// TIA Portal V20 export
// export: Created 2025-12-01T14:57:24.3574647Z, ExportSetting None, DisplayName Totally Integrated Automation Portal, DisplayVersion V20 Update 3, DisplayName TIA Portal Openness, DisplayVersion V20 Update 3, DisplayName TIA Portal Version Control Interface, DisplayVersion V20 Update 3, DisplayName STEP 7 Professional, DisplayVersion V20 Update 3, DisplayName STEP 7 Safety, DisplayVersion V20 Update 2, DisplayName WinCC Basic/Comfort/Advanced, DisplayVersion V20 Update 3, DisplayName WinCC Professional, DisplayVersion V20 Update 3, DisplayName WinCC Unified, DisplayVersion V20 Update 3
FUNCTION_BLOCK "FB20_M_PASO_E1E3_S1S3_2Puertas"   // FB20, LAD
TITLE = Control del Ramal de Salidas
{ S7_Optimized_Access := 'FALSE' }
AUTHOR : PASO
NAME : 20150327
VERSION : 3.3
// stored: AutoNumber false, SetENOAutomatically false
   VAR_INPUT
      Mesa : UInt;   // Mesa de la FB
      Error_Tx : Bool;
      EnTension : Bool;   // Existe Tension en la Mesa
      Termico_Tx : Bool;
      pHsMx_1 : Bool;   // Desactiva si Transferencia controlada
      pHsMx_2 : Bool;   // Desactiva si Transferencia controlada
      pHsMx_PR1 : Bool;   // pHs de Protrusion de la Mesa. Nota: No existe >> ON
      pHsMx_PR3 : Bool;   // pHs de Protrusion de la Mesa. Nota: No existe >> ON
      Avance_Tx : Bool;
      Retroceso_Tx : Bool;
      PUE1_Abierta : Bool;
      PUE1_Cerrada : Bool;
      PUE3_Abierta : Bool;
      PUE3_Cerrada : Bool;
      MAnt_DescargaAct_M1 : Bool;
      ATF_Ent_M1 : Bool;
      P_Mens_Ent_M1 : Bool;
      MAnt_DescargaAct_M3 : Bool;
      AVTF_Ent_M3 : Bool;
      P_Mens_Ent_M3 : Bool;
      PTF_Sal_M1 : Bool;
      FTF_Sal_M1 : Bool;
      PTF_Sal_M3 : Bool;
      FTF_Sal_M3 : Bool;
      Mx_VelocidadLenta_In : Bool;   // Forzar a Velociada Lenta
      F_EnvMens_Mx : Bool;
      OrdSal_S01 : Bool;
      OrdSal_S03 : Bool;
      V_CNT_pHsMx : Int := 300;
      V_CNT_pHsMx_FTF : Int := 50;   // Valor contador para FTF_Mant
      V_CNTSeg_pHsMx : Int := 2000;
      V_CNT_PasoLenta : Int := 2000;
      V_CNT_ApHsMx : Int := 500;
      V_CNTSeg_ApHsMx : Int := 2000;
      V_CNT_Simultaneo : Int := 1000;
      V_InicioSimultaneo : Int := 0;
      V_FinSimultaneo : Int := 0;
      V_TOut_Tx_Mx : Int := 30000;
      V_TOut_PUERTA : Int := 5000;
      V_TMP_Protrusion : Int := 200;   // TMP de Protrusion
      V_CNT_PerdidapHs : Int := 1000;
   END_VAR
   VAR_OUTPUT
      P_EnvMens_PMx : Bool;
      P_RecepOK_Mx : Bool;
      PTF_Ent_M1 : Bool;
      FTF_Ent_M1 : Bool;
      PTF_Ent_M3 : Bool;
      FTF_Ent_M3 : Bool;
      AVTF_Sal_M1 : Bool;
      P_Mens_Sal_M1 : Bool;
      AVTF_Sal_M3 : Bool;
      P_Mens_Sal_M3 : Bool;
   END_VAR
   VAR
      Anular_prE1 : Bool;   // ???
      Anular_prS3 : Bool;   // ???
      Mx_ET00 : Bool;
      Mx_ET01 : Bool;
      Mx_ET02 : Bool;
      Mx_ET08 : Bool;
      Mx_ET09 : Bool;
      Mx_ET10 : Bool;
      Mx_ET11 : Bool;
      Mx_ET12 : Bool;
      Mx_ET13 : Bool;
      Mx_ET50 : Bool;
      Mx_ET51 : Bool;
      Mx_ET110 : Bool;
      Mx_ET111 : Bool;
      Mx_ET150 : Bool;
      Mx_ET151 : Bool;
      Selec_M1_Entrada : Bool;
      Selec_M3_Entrada : Bool;
      Selec_M1_Salida : Bool;
      Selec_M3_Salida : Bool;
      MEnt_DescargaAct : Bool;
      AVTF_MEnt : Bool;
      P_Mens_MEnt : Bool;   // Interlock >> P_Mens de MAnt >> Mx
      PTF_MEnt : Bool;
      FTF_MEnt : Bool;
      AVTF_MSal : Bool;
      P_Mens_MSal : Bool;   // Interlock >> P_Mens de Mx >> MSig
      PTF_MSal : Bool;
      FTF_MSal : Bool;
      ProtocoloIniciado : Bool;
      CNT_pHsMx_FTF_OK : Bool;
      Simultaneo_Mx : Bool;
      STAT_EnvMens_PMx : Bool;
      MA_Abrir_PUE1 : Bool;
      MA_Cerrar_PUE1 : Bool;
      MA_Abrir_PUE3 : Bool;
      MA_Cerrar_PUE3 : Bool;
      CNT_pHsMx { S7_SetPoint := 'True'} : "FB910_CNT_UHS";
      CNTSeg_pHsMx { S7_SetPoint := 'True'} : "FB910_CNT_UHS";
      CNT_ApHsMx { S7_SetPoint := 'True'} : "FB910_CNT_UHS";
      CNTSeg_ApHsMx { S7_SetPoint := 'True'} : "FB910_CNT_UHS";
      CNT_Simultaneo { S7_SetPoint := 'True'} : "FB910_CNT_UHS";
      TMP_EnTension { S7_SetPoint := 'True'} : "FB910_CNT_UHS";
      TOut_Av_Mx { S7_SetPoint := 'True'} : "FB910_CNT_UHS";
      TOut_Ret_Mx { S7_SetPoint := 'True'} : "FB910_CNT_UHS";
      TOut_Abrir_PUE1 { S7_SetPoint := 'True'} : "FB910_CNT_UHS";
      TOut_Cerrar_PUE1 { S7_SetPoint := 'True'} : "FB910_CNT_UHS";
      TOut_Abrir_PUE3 { S7_SetPoint := 'True'} : "FB910_CNT_UHS";
      TOut_Cerrar_PUE3 { S7_SetPoint := 'True'} : "FB910_CNT_UHS";
      TMP_Protrusion { S7_SetPoint := 'True'} : "FB910_CNT_UHS";   // TMP de la Protrusion
      CNT_PerdidapHs { S7_SetPoint := 'True'} : "FB910_CNT_UHS";
   END_VAR
   VAR_TEMP
      EstadoZona : "EstadoZona";   // Estado de Zona de la Mesa
      EstadoVI : "EstadosMesa";   // Estado del Vehiculo Inteliguente de la Mesa
      ConfigFB : "UDT_ConfigFB";   // Configuracion de la FB de la Mesa
      V_Protrusion : Int;
      Aux_ET00 : Bool;
   END_VAR
   VAR_TEMP   // added for the SCL form of the ladder/FBD networks
      _w1 : Bool;
      _w2 : Bool;
   END_VAR
BEGIN

REGION Network 1: INICIALIZAR - Recoger las Variables de Estado de la Mesa
   // Se recoge - Estado_CBx
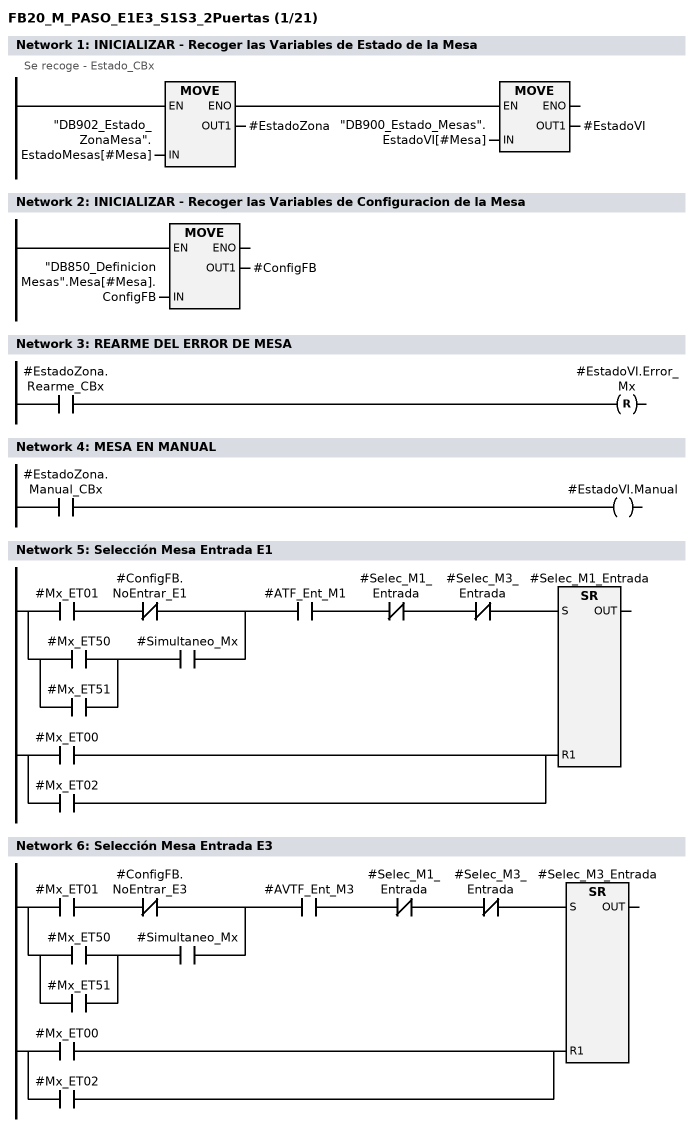
   RUNG wire#powerrail
      Move(in := "DB902_Estado_ZonaMesa".EstadoMesas[#Mesa], out1 => #EstadoZona)
      Move(in := "DB900_Estado_Mesas".EstadoVI[#Mesa], out1 => #EstadoVI)
   END_RUNG
   // the same network as SCL:
   #EstadoZona := "DB902_Estado_ZonaMesa".EstadoMesas[#Mesa];
   #EstadoVI := "DB900_Estado_Mesas".EstadoVI[#Mesa];
END_REGION

REGION Network 2: INICIALIZAR - Recoger las Variables de Configuracion de la Mesa
   RUNG wire#powerrail
      Move(in := "DB850_DefinicionMesas".Mesa[#Mesa].ConfigFB, out1 => #ConfigFB)
   END_RUNG
   // the same network as SCL:
   #ConfigFB := "DB850_DefinicionMesas".Mesa[#Mesa].ConfigFB;
END_REGION

REGION Network 3: REARME DEL ERROR DE MESA
   RUNG wire#powerrail
      Contact( #EstadoZona.Rearme_CBx )
      R_Coil( #EstadoVI.Error_Mx )
   END_RUNG
   // the same network as SCL:
   IF #EstadoZona.Rearme_CBx THEN #EstadoVI.Error_Mx := FALSE; END_IF;
END_REGION

REGION Network 4: MESA EN MANUAL
   RUNG wire#powerrail
      Contact( #EstadoZona.Manual_CBx )
      Coil( #EstadoVI.Manual )
   END_RUNG
   // the same network as SCL:
   #EstadoVI.Manual := #EstadoZona.Manual_CBx;
END_REGION

REGION Network 5: Selección Mesa Entrada E1
   RUNG wire#powerrail
      Contact( #Mx_ET01 )
      I_Contact( #ConfigFB.NoEntrar_E1 )
      wire#w1
      Contact( #ATF_Ent_M1 )
      I_Contact( #Selec_M1_Entrada )
      I_Contact( #Selec_M3_Entrada )
      S_SR(operand := #Selec_M1_Entrada, r1 := wire#w3)
   END_RUNG
   RUNG wire#powerrail
      Contact( #Mx_ET50 )
      wire#w2
      Contact( #Simultaneo_Mx )
   END_RUNG wire#w1
   RUNG wire#powerrail
      Contact( #Mx_ET51 )
   END_RUNG wire#w2
   RUNG wire#powerrail
      Contact( #Mx_ET00 )
   END_RUNG wire#w3
   RUNG wire#powerrail
      Contact( #Mx_ET02 )
   END_RUNG wire#w3
   // the same network as SCL:
   IF ((#Mx_ET01 AND NOT #ConfigFB.NoEntrar_E1) OR ((#Mx_ET50 OR #Mx_ET51) AND #Simultaneo_Mx)) AND #ATF_Ent_M1 AND NOT #Selec_M1_Entrada AND NOT #Selec_M3_Entrada THEN
       #Selec_M1_Entrada := TRUE;   // SR flip-flop
   END_IF;
   IF #Mx_ET00 OR #Mx_ET02 THEN #Selec_M1_Entrada := FALSE; END_IF;
END_REGION

REGION Network 6: Selección Mesa Entrada E3
   RUNG wire#powerrail
      Contact( #Mx_ET01 )
      I_Contact( #ConfigFB.NoEntrar_E3 )
      wire#w1
      Contact( #AVTF_Ent_M3 )
      I_Contact( #Selec_M1_Entrada )
      I_Contact( #Selec_M3_Entrada )
      S_SR(operand := #Selec_M3_Entrada, r1 := wire#w3)
   END_RUNG
   RUNG wire#powerrail
      Contact( #Mx_ET50 )
      wire#w2
      Contact( #Simultaneo_Mx )
   END_RUNG wire#w1
   RUNG wire#powerrail
      Contact( #Mx_ET51 )
   END_RUNG wire#w2
   RUNG wire#powerrail
      Contact( #Mx_ET00 )
   END_RUNG wire#w3
   RUNG wire#powerrail
      Contact( #Mx_ET02 )
   END_RUNG wire#w3
   // the same network as SCL:
   IF ((#Mx_ET01 AND NOT #ConfigFB.NoEntrar_E3) OR ((#Mx_ET50 OR #Mx_ET51) AND #Simultaneo_Mx)) AND #AVTF_Ent_M3 AND NOT #Selec_M1_Entrada AND NOT #Selec_M3_Entrada THEN
       #Selec_M3_Entrada := TRUE;   // SR flip-flop
   END_IF;
   IF #Mx_ET00 OR #Mx_ET02 THEN #Selec_M3_Entrada := FALSE; END_IF;
END_REGION

REGION Network 7: Selección Mesa Salida S1
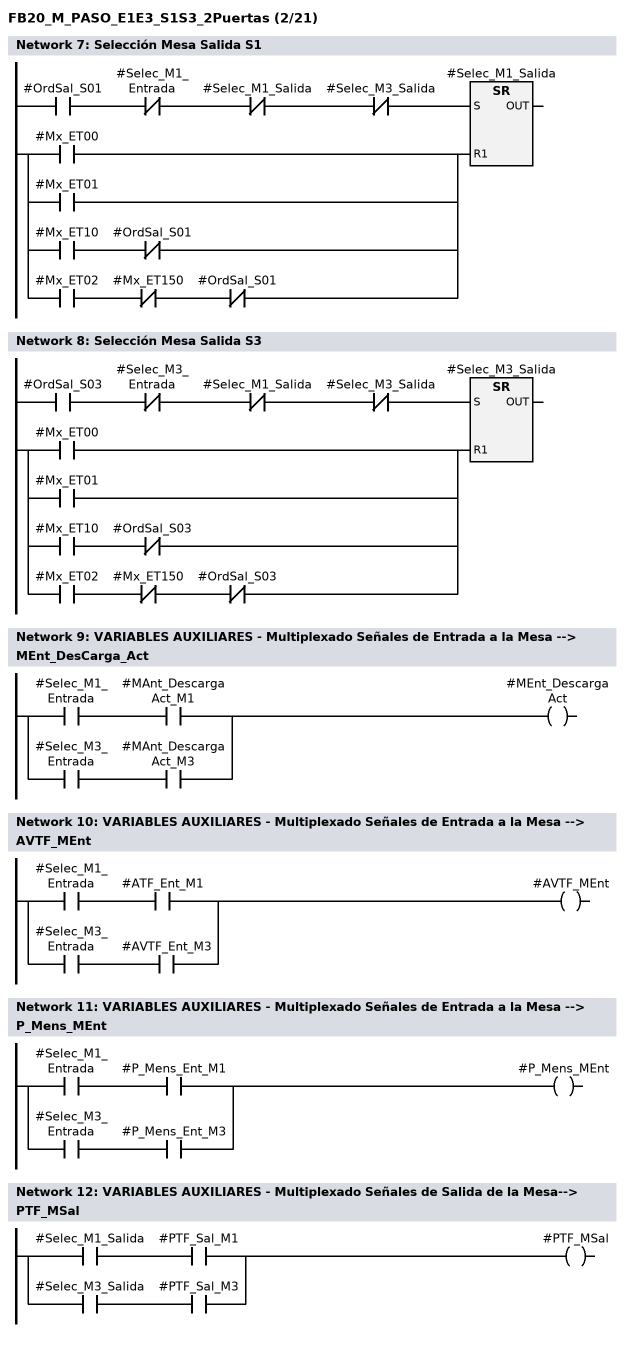
   RUNG wire#powerrail
      Contact( #OrdSal_S01 )
      I_Contact( #Selec_M1_Entrada )
      I_Contact( #Selec_M1_Salida )
      I_Contact( #Selec_M3_Salida )
      S_SR(operand := #Selec_M1_Salida, r1 := wire#w1)
   END_RUNG
   RUNG wire#powerrail
      Contact( #Mx_ET00 )
   END_RUNG wire#w1
   RUNG wire#powerrail
      Contact( #Mx_ET01 )
   END_RUNG wire#w1
   RUNG wire#powerrail
      Contact( #Mx_ET10 )
      I_Contact( #OrdSal_S01 )
   END_RUNG wire#w1
   RUNG wire#powerrail
      Contact( #Mx_ET02 )
      I_Contact( #Mx_ET150 )
      I_Contact( #OrdSal_S01 )
   END_RUNG wire#w1
   // the same network as SCL:
   IF #OrdSal_S01 AND NOT #Selec_M1_Entrada AND NOT #Selec_M1_Salida AND NOT #Selec_M3_Salida THEN
       #Selec_M1_Salida := TRUE;   // SR flip-flop
   END_IF;
   IF #Mx_ET00 OR #Mx_ET01 OR (#Mx_ET10 AND NOT #OrdSal_S01) OR (#Mx_ET02 AND NOT #Mx_ET150 AND NOT #OrdSal_S01) THEN
       #Selec_M1_Salida := FALSE;
   END_IF;
END_REGION

REGION Network 8: Selección Mesa Salida S3
   RUNG wire#powerrail
      Contact( #OrdSal_S03 )
      I_Contact( #Selec_M3_Entrada )
      I_Contact( #Selec_M1_Salida )
      I_Contact( #Selec_M3_Salida )
      S_SR(operand := #Selec_M3_Salida, r1 := wire#w1)
   END_RUNG
   RUNG wire#powerrail
      Contact( #Mx_ET00 )
   END_RUNG wire#w1
   RUNG wire#powerrail
      Contact( #Mx_ET01 )
   END_RUNG wire#w1
   RUNG wire#powerrail
      Contact( #Mx_ET10 )
      I_Contact( #OrdSal_S03 )
   END_RUNG wire#w1
   RUNG wire#powerrail
      Contact( #Mx_ET02 )
      I_Contact( #Mx_ET150 )
      I_Contact( #OrdSal_S03 )
   END_RUNG wire#w1
   // the same network as SCL:
   IF #OrdSal_S03 AND NOT #Selec_M3_Entrada AND NOT #Selec_M1_Salida AND NOT #Selec_M3_Salida THEN
       #Selec_M3_Salida := TRUE;   // SR flip-flop
   END_IF;
   IF #Mx_ET00 OR #Mx_ET01 OR (#Mx_ET10 AND NOT #OrdSal_S03) OR (#Mx_ET02 AND NOT #Mx_ET150 AND NOT #OrdSal_S03) THEN
       #Selec_M3_Salida := FALSE;
   END_IF;
END_REGION

REGION Network 9: VARIABLES AUXILIARES - Multiplexado Señales de Entrada a la Mesa --> MEnt_DesCarga_Act
   RUNG wire#powerrail
      Contact( #Selec_M1_Entrada )
      Contact( #MAnt_DescargaAct_M1 )
      wire#w1
      Coil( #MEnt_DescargaAct )
   END_RUNG
   RUNG wire#powerrail
      Contact( #Selec_M3_Entrada )
      Contact( #MAnt_DescargaAct_M3 )
   END_RUNG wire#w1
   // the same network as SCL:
   #MEnt_DescargaAct := (#Selec_M1_Entrada AND #MAnt_DescargaAct_M1) OR (#Selec_M3_Entrada AND #MAnt_DescargaAct_M3);
END_REGION

REGION Network 10: VARIABLES AUXILIARES - Multiplexado Señales de Entrada a la Mesa --> AVTF_MEnt
   RUNG wire#powerrail
      Contact( #Selec_M1_Entrada )
      Contact( #ATF_Ent_M1 )
      wire#w1
      Coil( #AVTF_MEnt )
   END_RUNG
   RUNG wire#powerrail
      Contact( #Selec_M3_Entrada )
      Contact( #AVTF_Ent_M3 )
   END_RUNG wire#w1
   // the same network as SCL:
   #AVTF_MEnt := (#Selec_M1_Entrada AND #ATF_Ent_M1) OR (#Selec_M3_Entrada AND #AVTF_Ent_M3);
END_REGION

REGION Network 11: VARIABLES AUXILIARES - Multiplexado Señales de Entrada a la Mesa --> P_Mens_MEnt
   RUNG wire#powerrail
      Contact( #Selec_M1_Entrada )
      Contact( #P_Mens_Ent_M1 )
      wire#w1
      Coil( #P_Mens_MEnt )
   END_RUNG
   RUNG wire#powerrail
      Contact( #Selec_M3_Entrada )
      Contact( #P_Mens_Ent_M3 )
   END_RUNG wire#w1
   // the same network as SCL:
   #P_Mens_MEnt := (#Selec_M1_Entrada AND #P_Mens_Ent_M1) OR (#Selec_M3_Entrada AND #P_Mens_Ent_M3);
END_REGION

REGION Network 12: VARIABLES AUXILIARES - Multiplexado Señales de Salida de la Mesa--> PTF_MSal
   RUNG wire#powerrail
      Contact( #Selec_M1_Salida )
      Contact( #PTF_Sal_M1 )
      wire#w1
      Coil( #PTF_MSal )
   END_RUNG
   RUNG wire#powerrail
      Contact( #Selec_M3_Salida )
      Contact( #PTF_Sal_M3 )
   END_RUNG wire#w1
   // the same network as SCL:
   #PTF_MSal := (#Selec_M1_Salida AND #PTF_Sal_M1) OR (#Selec_M3_Salida AND #PTF_Sal_M3);
END_REGION

REGION Network 13: VARIABLES AUXILIARES - Multiplexado Señales de Salida de la Mesa--> FTF_MSal
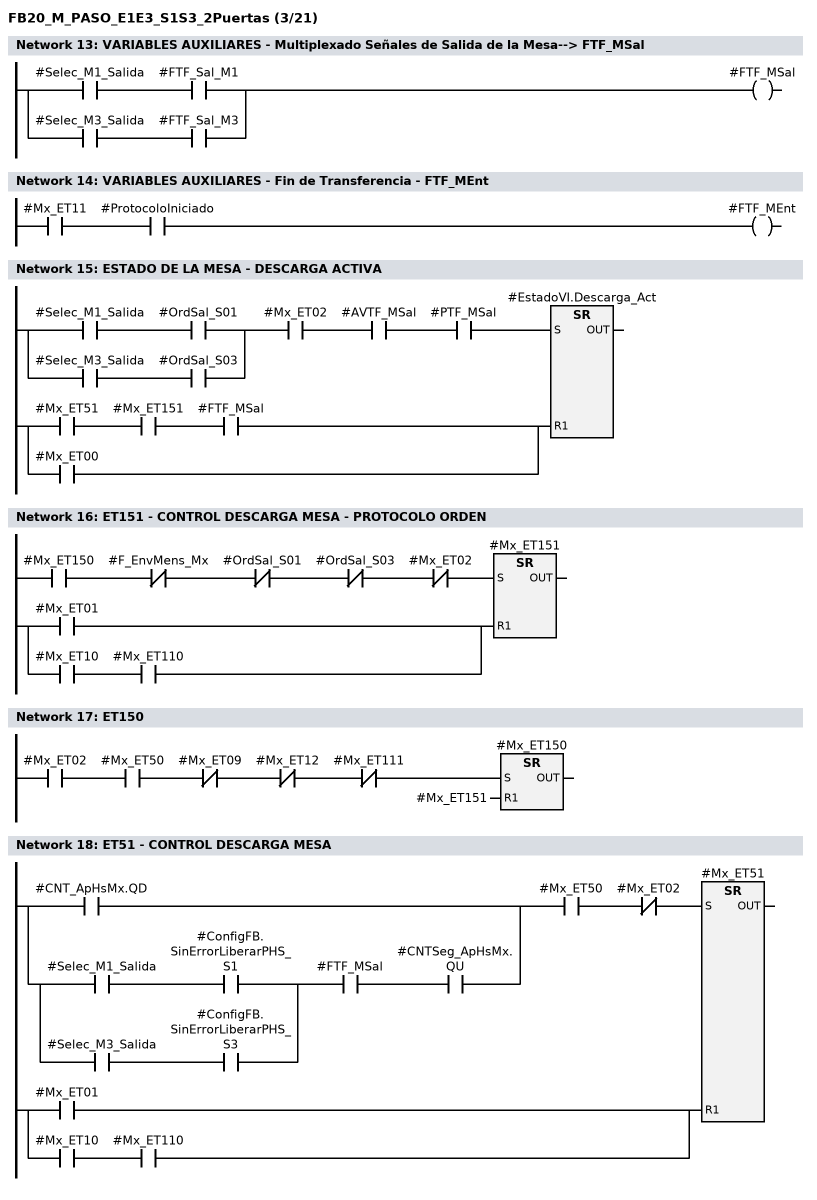
   RUNG wire#powerrail
      Contact( #Selec_M1_Salida )
      Contact( #FTF_Sal_M1 )
      wire#w1
      Coil( #FTF_MSal )
   END_RUNG
   RUNG wire#powerrail
      Contact( #Selec_M3_Salida )
      Contact( #FTF_Sal_M3 )
   END_RUNG wire#w1
   // the same network as SCL:
   #FTF_MSal := (#Selec_M1_Salida AND #FTF_Sal_M1) OR (#Selec_M3_Salida AND #FTF_Sal_M3);
END_REGION

REGION Network 14: VARIABLES AUXILIARES - Fin de Transferencia - FTF_MEnt
   RUNG wire#powerrail
      Contact( #Mx_ET11 )
      Contact( #ProtocoloIniciado )
      Coil( #FTF_MEnt )
   END_RUNG
   // the same network as SCL:
   #FTF_MEnt := #Mx_ET11 AND #ProtocoloIniciado;
END_REGION

REGION Network 15: ESTADO DE LA MESA - DESCARGA ACTIVA
   RUNG wire#powerrail
      Contact( #Selec_M1_Salida )
      Contact( #OrdSal_S01 )
      wire#w1
      Contact( #Mx_ET02 )
      Contact( #AVTF_MSal )
      Contact( #PTF_MSal )
      S_SR(operand := #EstadoVI.Descarga_Act, r1 := wire#w2)
   END_RUNG
   RUNG wire#powerrail
      Contact( #Selec_M3_Salida )
      Contact( #OrdSal_S03 )
   END_RUNG wire#w1
   RUNG wire#powerrail
      Contact( #Mx_ET51 )
      Contact( #Mx_ET151 )
      Contact( #FTF_MSal )
   END_RUNG wire#w2
   RUNG wire#powerrail
      Contact( #Mx_ET00 )
   END_RUNG wire#w2
   // the same network as SCL:
   IF ((#Selec_M1_Salida AND #OrdSal_S01) OR (#Selec_M3_Salida AND #OrdSal_S03)) AND #Mx_ET02 AND #AVTF_MSal AND #PTF_MSal THEN
       #EstadoVI.Descarga_Act := TRUE;   // SR flip-flop
   END_IF;
   IF (#Mx_ET51 AND #Mx_ET151 AND #FTF_MSal) OR #Mx_ET00 THEN #EstadoVI.Descarga_Act := FALSE; END_IF;
END_REGION

REGION Network 16: ET151 - CONTROL DESCARGA MESA - PROTOCOLO ORDEN
   RUNG wire#powerrail
      Contact( #Mx_ET150 )
      I_Contact( #F_EnvMens_Mx )
      I_Contact( #OrdSal_S01 )
      I_Contact( #OrdSal_S03 )
      I_Contact( #Mx_ET02 )
      S_SR(operand := #Mx_ET151, r1 := wire#w1)
   END_RUNG
   RUNG wire#powerrail
      Contact( #Mx_ET01 )
   END_RUNG wire#w1
   RUNG wire#powerrail
      Contact( #Mx_ET10 )
      Contact( #Mx_ET110 )
   END_RUNG wire#w1
   // the same network as SCL:
   IF #Mx_ET150 AND NOT #F_EnvMens_Mx AND NOT #OrdSal_S01 AND NOT #OrdSal_S03 AND NOT #Mx_ET02 THEN
       #Mx_ET151 := TRUE;   // SR flip-flop
   END_IF;
   IF #Mx_ET01 OR (#Mx_ET10 AND #Mx_ET110) THEN #Mx_ET151 := FALSE; END_IF;
END_REGION

REGION Network 17: ET150
   RUNG wire#powerrail
      Contact( #Mx_ET02 )
      Contact( #Mx_ET50 )
      I_Contact( #Mx_ET09 )
      I_Contact( #Mx_ET12 )
      I_Contact( #Mx_ET111 )
      S_SR(operand := #Mx_ET150, r1 := #Mx_ET151)
   END_RUNG
   // the same network as SCL:
   IF #Mx_ET02 AND #Mx_ET50 AND NOT #Mx_ET09 AND NOT #Mx_ET12 AND NOT #Mx_ET111 THEN
       #Mx_ET150 := TRUE;   // SR flip-flop
   END_IF;
   IF #Mx_ET151 THEN #Mx_ET150 := FALSE; END_IF;
END_REGION

REGION Network 18: ET51 - CONTROL DESCARGA MESA
   RUNG wire#powerrail
      Contact( #CNT_ApHsMx.QD )
      wire#w1
      Contact( #Mx_ET50 )
      I_Contact( #Mx_ET02 )
      S_SR(operand := #Mx_ET51, r1 := wire#w3)
   END_RUNG
   RUNG wire#powerrail
      Contact( #Selec_M1_Salida )
      Contact( #ConfigFB.SinErrorLiberarPHS_S1 )
      wire#w2
      Contact( #FTF_MSal )
      Contact( #CNTSeg_ApHsMx.QU )
   END_RUNG wire#w1
   RUNG wire#powerrail
      Contact( #Selec_M3_Salida )
      Contact( #ConfigFB.SinErrorLiberarPHS_S3 )
   END_RUNG wire#w2
   RUNG wire#powerrail
      Contact( #Mx_ET01 )
   END_RUNG wire#w3
   RUNG wire#powerrail
      Contact( #Mx_ET10 )
      Contact( #Mx_ET110 )
   END_RUNG wire#w3
   // the same network as SCL:
   IF (#CNT_ApHsMx.QD OR (((#Selec_M1_Salida AND #ConfigFB.SinErrorLiberarPHS_S1) OR (#Selec_M3_Salida AND #ConfigFB.SinErrorLiberarPHS_S3)) AND #FTF_MSal AND #CNTSeg_ApHsMx.QU)) AND #Mx_ET50 AND NOT #Mx_ET02 THEN
       #Mx_ET51 := TRUE;   // SR flip-flop
   END_IF;
   IF #Mx_ET01 OR (#Mx_ET10 AND #Mx_ET110) THEN #Mx_ET51 := FALSE; END_IF;
END_REGION

REGION Network 19: ET50
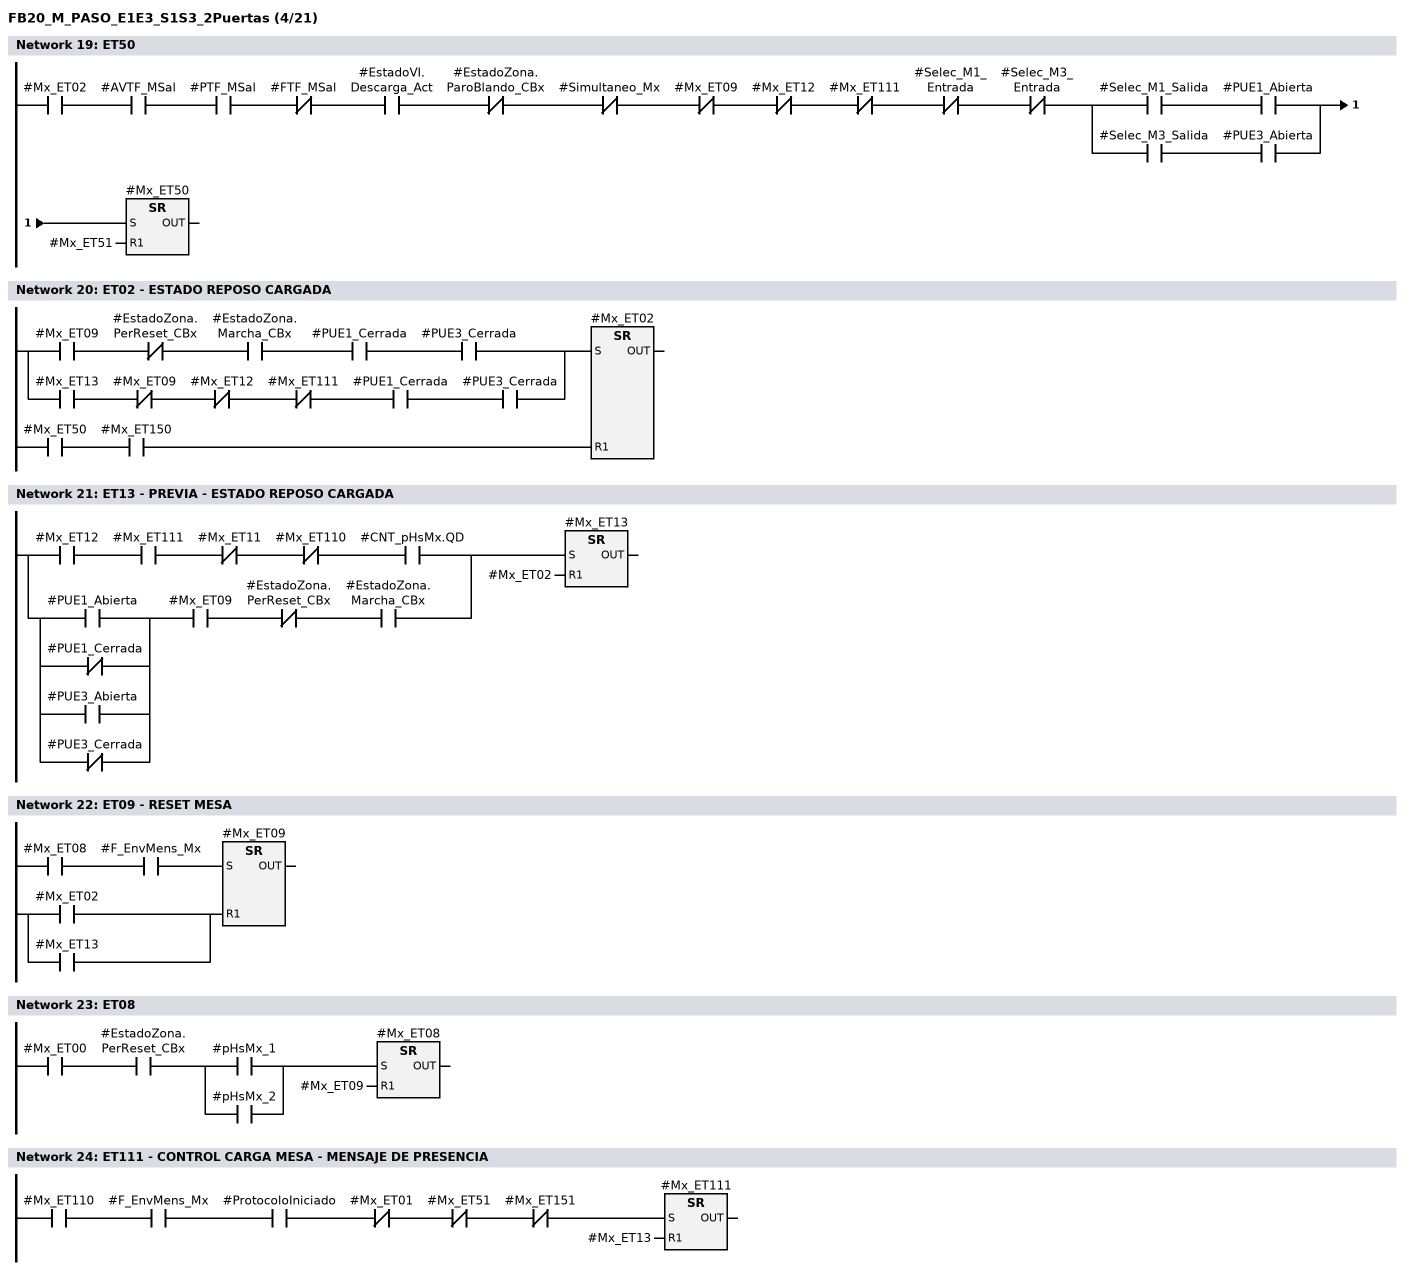
   RUNG wire#powerrail
      Contact( #Mx_ET02 )
      Contact( #AVTF_MSal )
      Contact( #PTF_MSal )
      I_Contact( #FTF_MSal )
      Contact( #EstadoVI.Descarga_Act )
      I_Contact( #EstadoZona.ParoBlando_CBx )
      I_Contact( #Simultaneo_Mx )
      I_Contact( #Mx_ET09 )
      I_Contact( #Mx_ET12 )
      I_Contact( #Mx_ET111 )
      I_Contact( #Selec_M1_Entrada )
      I_Contact( #Selec_M3_Entrada )
      wire#w1
      Contact( #Selec_M1_Salida )
      Contact( #PUE1_Abierta )
      wire#w2
      S_SR(operand := #Mx_ET50, r1 := #Mx_ET51)
   END_RUNG
   RUNG wire#w1
      Contact( #Selec_M3_Salida )
      Contact( #PUE3_Abierta )
   END_RUNG wire#w2
   // the same network as SCL:
   IF #Mx_ET02 AND #AVTF_MSal AND #PTF_MSal AND NOT #FTF_MSal AND #EstadoVI.Descarga_Act AND NOT #EstadoZona.ParoBlando_CBx AND NOT #Simultaneo_Mx AND NOT #Mx_ET09 AND NOT #Mx_ET12 AND NOT #Mx_ET111 AND NOT #Selec_M1_Entrada AND NOT #Selec_M3_Entrada AND ((#Selec_M1_Salida AND #PUE1_Abierta) OR (#Selec_M3_Salida AND #PUE3_Abierta)) THEN
       #Mx_ET50 := TRUE;   // SR flip-flop
   END_IF;
   IF #Mx_ET51 THEN #Mx_ET50 := FALSE; END_IF;
END_REGION

REGION Network 20: ET02 - ESTADO REPOSO CARGADA
   RUNG wire#powerrail
      Contact( #Mx_ET09 )
      I_Contact( #EstadoZona.PerReset_CBx )
      Contact( #EstadoZona.Marcha_CBx )
      Contact( #PUE1_Cerrada )
      Contact( #PUE3_Cerrada )
      wire#w1
      S_SR(operand := #Mx_ET02, r1 := wire#w2)
   END_RUNG
   RUNG wire#powerrail
      Contact( #Mx_ET13 )
      I_Contact( #Mx_ET09 )
      I_Contact( #Mx_ET12 )
      I_Contact( #Mx_ET111 )
      Contact( #PUE1_Cerrada )
      Contact( #PUE3_Cerrada )
   END_RUNG wire#w1
   RUNG wire#powerrail
      Contact( #Mx_ET50 )
      Contact( #Mx_ET150 )
   END_RUNG wire#w2
   // the same network as SCL:
   IF (#Mx_ET09 AND NOT #EstadoZona.PerReset_CBx AND #EstadoZona.Marcha_CBx AND #PUE1_Cerrada AND #PUE3_Cerrada) OR (#Mx_ET13 AND NOT #Mx_ET09 AND NOT #Mx_ET12 AND NOT #Mx_ET111 AND #PUE1_Cerrada AND #PUE3_Cerrada) THEN
       #Mx_ET02 := TRUE;   // SR flip-flop
   END_IF;
   IF #Mx_ET50 AND #Mx_ET150 THEN #Mx_ET02 := FALSE; END_IF;
END_REGION

REGION Network 21: ET13 - PREVIA - ESTADO REPOSO CARGADA
   RUNG wire#powerrail
      Contact( #Mx_ET12 )
      Contact( #Mx_ET111 )
      I_Contact( #Mx_ET11 )
      I_Contact( #Mx_ET110 )
      Contact( #CNT_pHsMx.QD )
      wire#w1
      S_SR(operand := #Mx_ET13, r1 := #Mx_ET02)
   END_RUNG
   RUNG wire#powerrail
      Contact( #PUE1_Abierta )
      wire#w2
      Contact( #Mx_ET09 )
      I_Contact( #EstadoZona.PerReset_CBx )
      Contact( #EstadoZona.Marcha_CBx )
   END_RUNG wire#w1
   RUNG wire#powerrail
      I_Contact( #PUE1_Cerrada )
   END_RUNG wire#w2
   RUNG wire#powerrail
      Contact( #PUE3_Abierta )
   END_RUNG wire#w2
   RUNG wire#powerrail
      I_Contact( #PUE3_Cerrada )
   END_RUNG wire#w2
   // the same network as SCL:
   IF (#Mx_ET12 AND #Mx_ET111 AND NOT #Mx_ET11 AND NOT #Mx_ET110 AND #CNT_pHsMx.QD) OR ((#PUE1_Abierta OR NOT #PUE1_Cerrada OR #PUE3_Abierta OR NOT #PUE3_Cerrada) AND #Mx_ET09 AND NOT #EstadoZona.PerReset_CBx AND #EstadoZona.Marcha_CBx) THEN
       #Mx_ET13 := TRUE;   // SR flip-flop
   END_IF;
   IF #Mx_ET02 THEN #Mx_ET13 := FALSE; END_IF;
END_REGION

REGION Network 22: ET09 - RESET MESA
   RUNG wire#powerrail
      Contact( #Mx_ET08 )
      Contact( #F_EnvMens_Mx )
      S_SR(operand := #Mx_ET09, r1 := wire#w1)
   END_RUNG
   RUNG wire#powerrail
      Contact( #Mx_ET02 )
   END_RUNG wire#w1
   RUNG wire#powerrail
      Contact( #Mx_ET13 )
   END_RUNG wire#w1
   // the same network as SCL:
   IF #Mx_ET08 AND #F_EnvMens_Mx THEN
       #Mx_ET09 := TRUE;   // SR flip-flop
   END_IF;
   IF #Mx_ET02 OR #Mx_ET13 THEN #Mx_ET09 := FALSE; END_IF;
END_REGION

REGION Network 23: ET08
   RUNG wire#powerrail
      Contact( #Mx_ET00 )
      Contact( #EstadoZona.PerReset_CBx )
      wire#w1
      Contact( #pHsMx_1 )
      wire#w2
      S_SR(operand := #Mx_ET08, r1 := #Mx_ET09)
   END_RUNG
   RUNG wire#w1
      Contact( #pHsMx_2 )
   END_RUNG wire#w2
   // the same network as SCL:
   IF #Mx_ET00 AND #EstadoZona.PerReset_CBx AND (#pHsMx_1 OR #pHsMx_2) THEN
       #Mx_ET08 := TRUE;   // SR flip-flop
   END_IF;
   IF #Mx_ET09 THEN #Mx_ET08 := FALSE; END_IF;
END_REGION

REGION Network 24: ET111 - CONTROL CARGA MESA - MENSAJE DE PRESENCIA
   RUNG wire#powerrail
      Contact( #Mx_ET110 )
      Contact( #F_EnvMens_Mx )
      Contact( #ProtocoloIniciado )
      I_Contact( #Mx_ET01 )
      I_Contact( #Mx_ET51 )
      I_Contact( #Mx_ET151 )
      S_SR(operand := #Mx_ET111, r1 := #Mx_ET13)
   END_RUNG
   // the same network as SCL:
   IF #Mx_ET110 AND #F_EnvMens_Mx AND #ProtocoloIniciado AND NOT #Mx_ET01 AND NOT #Mx_ET51 AND NOT #Mx_ET151 THEN
       #Mx_ET111 := TRUE;   // SR flip-flop
   END_IF;
   IF #Mx_ET13 THEN #Mx_ET111 := FALSE; END_IF;
END_REGION

REGION Network 25: ET110
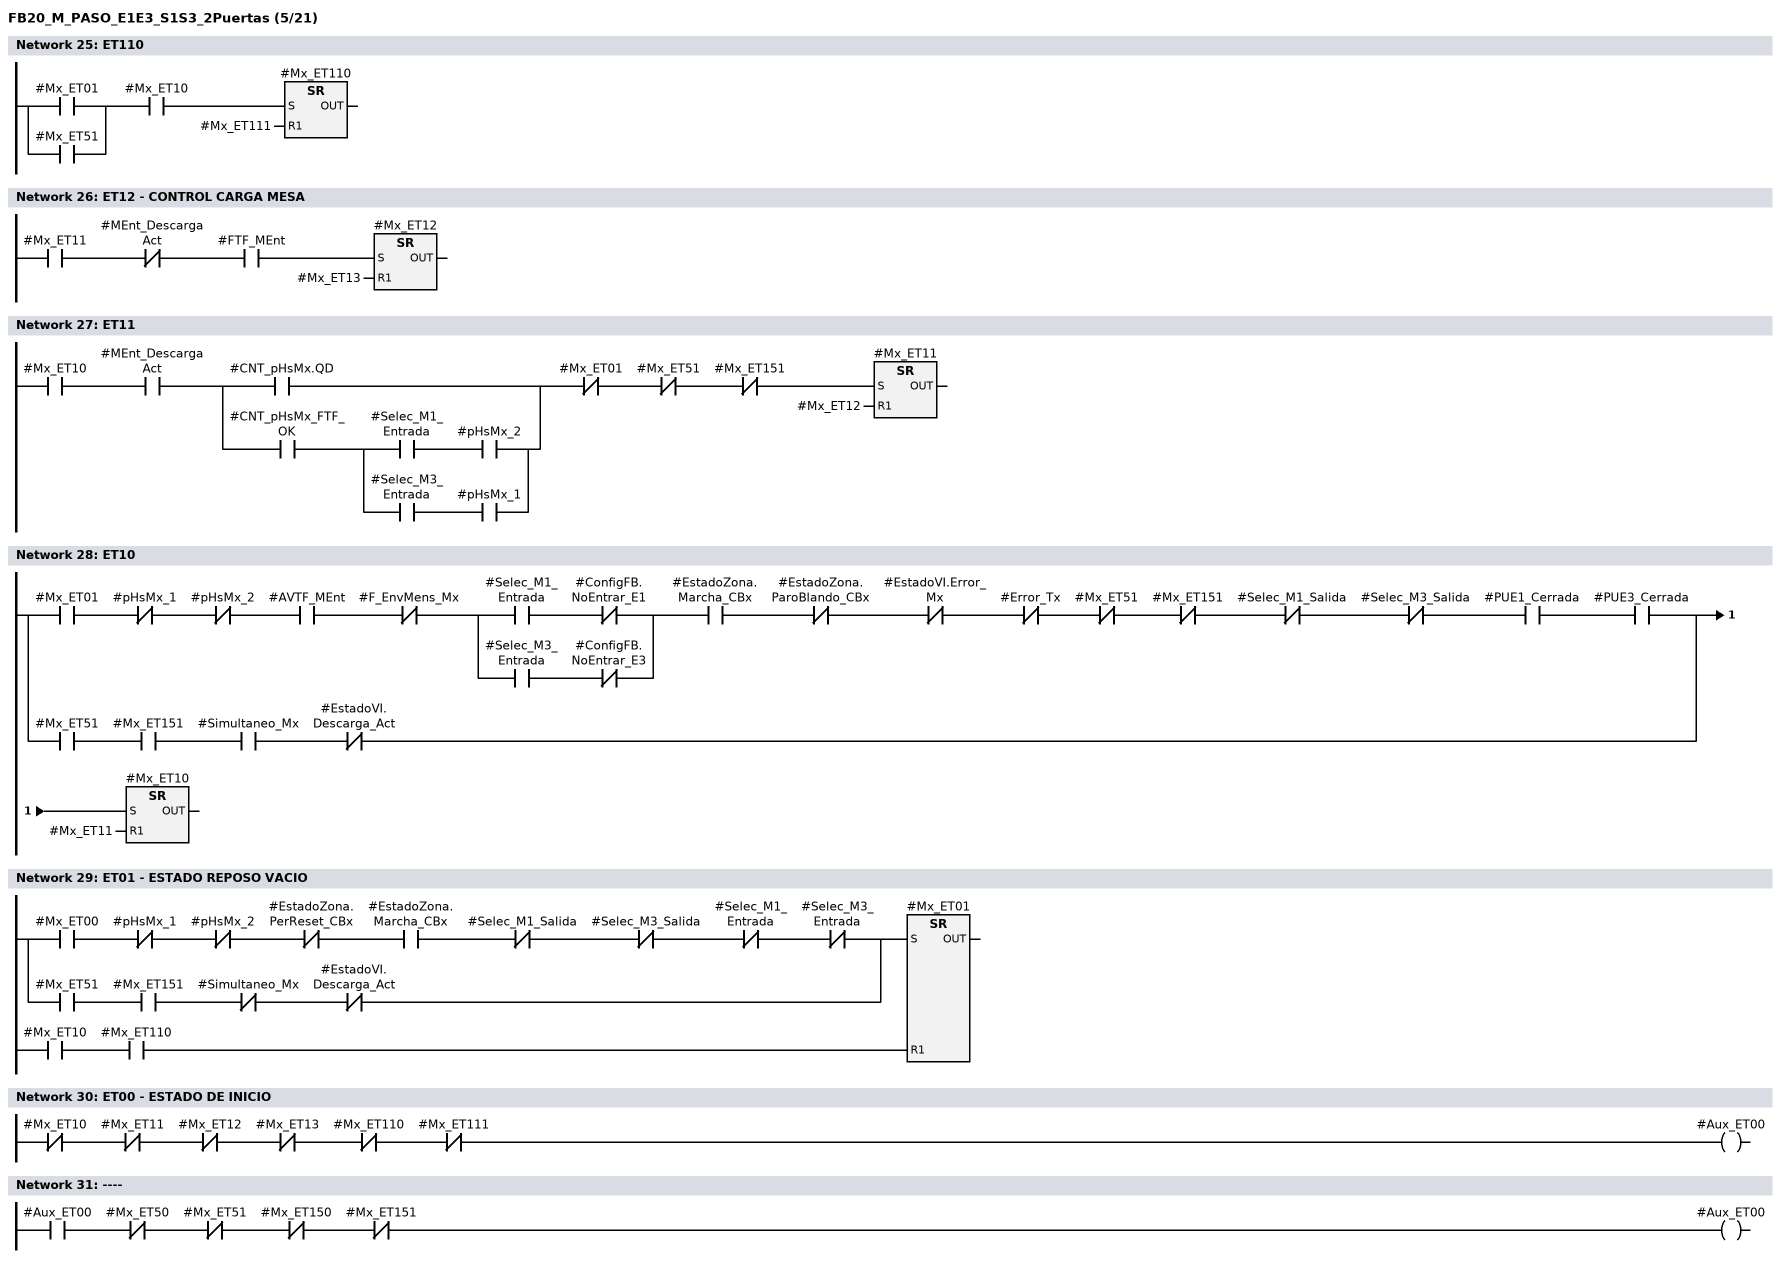
   RUNG wire#powerrail
      Contact( #Mx_ET01 )
      wire#w1
      Contact( #Mx_ET10 )
      S_SR(operand := #Mx_ET110, r1 := #Mx_ET111)
   END_RUNG
   RUNG wire#powerrail
      Contact( #Mx_ET51 )
   END_RUNG wire#w1
   // the same network as SCL:
   IF (#Mx_ET01 OR #Mx_ET51) AND #Mx_ET10 THEN
       #Mx_ET110 := TRUE;   // SR flip-flop
   END_IF;
   IF #Mx_ET111 THEN #Mx_ET110 := FALSE; END_IF;
END_REGION

REGION Network 26: ET12 - CONTROL CARGA MESA
   RUNG wire#powerrail
      Contact( #Mx_ET11 )
      I_Contact( #MEnt_DescargaAct )
      Contact( #FTF_MEnt )
      S_SR(operand := #Mx_ET12, r1 := #Mx_ET13)
   END_RUNG
   // the same network as SCL:
   IF #Mx_ET11 AND NOT #MEnt_DescargaAct AND #FTF_MEnt THEN
       #Mx_ET12 := TRUE;   // SR flip-flop
   END_IF;
   IF #Mx_ET13 THEN #Mx_ET12 := FALSE; END_IF;
END_REGION

REGION Network 27: ET11
   RUNG wire#powerrail
      Contact( #Mx_ET10 )
      Contact( #MEnt_DescargaAct )
      wire#w1
      Contact( #CNT_pHsMx.QD )
      wire#w2
      I_Contact( #Mx_ET01 )
      I_Contact( #Mx_ET51 )
      I_Contact( #Mx_ET151 )
      S_SR(operand := #Mx_ET11, r1 := #Mx_ET12)
   END_RUNG
   RUNG wire#w1
      Contact( #CNT_pHsMx_FTF_OK )
      wire#w3
      Contact( #Selec_M1_Entrada )
      Contact( #pHsMx_2 )
   END_RUNG wire#w2
   RUNG wire#w3
      Contact( #Selec_M3_Entrada )
      Contact( #pHsMx_1 )
   END_RUNG wire#w2
   // the same network as SCL:
   IF #Mx_ET10 AND #MEnt_DescargaAct AND (#CNT_pHsMx.QD OR (#CNT_pHsMx_FTF_OK AND ((#Selec_M1_Entrada AND #pHsMx_2) OR (#Selec_M3_Entrada AND #pHsMx_1)))) AND NOT #Mx_ET01 AND NOT #Mx_ET51 AND NOT #Mx_ET151 THEN
       #Mx_ET11 := TRUE;   // SR flip-flop
   END_IF;
   IF #Mx_ET12 THEN #Mx_ET11 := FALSE; END_IF;
END_REGION

REGION Network 28: ET10
   RUNG wire#powerrail
      Contact( #Mx_ET01 )
      I_Contact( #pHsMx_1 )
      I_Contact( #pHsMx_2 )
      Contact( #AVTF_MEnt )
      I_Contact( #F_EnvMens_Mx )
      wire#w1
      Contact( #Selec_M1_Entrada )
      I_Contact( #ConfigFB.NoEntrar_E1 )
      wire#w2
      Contact( #EstadoZona.Marcha_CBx )
      I_Contact( #EstadoZona.ParoBlando_CBx )
      I_Contact( #EstadoVI.Error_Mx )
      I_Contact( #Error_Tx )
      I_Contact( #Mx_ET51 )
      I_Contact( #Mx_ET151 )
      I_Contact( #Selec_M1_Salida )
      I_Contact( #Selec_M3_Salida )
      Contact( #PUE1_Cerrada )
      Contact( #PUE3_Cerrada )
      wire#w3
      S_SR(operand := #Mx_ET10, r1 := #Mx_ET11)
   END_RUNG
   RUNG wire#w1
      Contact( #Selec_M3_Entrada )
      I_Contact( #ConfigFB.NoEntrar_E3 )
   END_RUNG wire#w2
   RUNG wire#powerrail
      Contact( #Mx_ET51 )
      Contact( #Mx_ET151 )
      Contact( #Simultaneo_Mx )
      I_Contact( #EstadoVI.Descarga_Act )
   END_RUNG wire#w3
   // the same network as SCL:
   IF (#Mx_ET01 AND NOT #pHsMx_1 AND NOT #pHsMx_2 AND #AVTF_MEnt AND NOT #F_EnvMens_Mx AND ((#Selec_M1_Entrada AND NOT #ConfigFB.NoEntrar_E1) OR (#Selec_M3_Entrada AND NOT #ConfigFB.NoEntrar_E3)) AND #EstadoZona.Marcha_CBx AND NOT #EstadoZona.ParoBlando_CBx AND NOT #EstadoVI.Error_Mx AND NOT #Error_Tx AND NOT #Mx_ET51 AND NOT #Mx_ET151 AND NOT #Selec_M1_Salida AND NOT #Selec_M3_Salida AND #PUE1_Cerrada AND #PUE3_Cerrada) OR (#Mx_ET51 AND #Mx_ET151 AND #Simultaneo_Mx AND NOT #EstadoVI.Descarga_Act) THEN
       #Mx_ET10 := TRUE;   // SR flip-flop
   END_IF;
   IF #Mx_ET11 THEN #Mx_ET10 := FALSE; END_IF;
END_REGION

REGION Network 29: ET01 - ESTADO REPOSO VACIO
   RUNG wire#powerrail
      Contact( #Mx_ET00 )
      I_Contact( #pHsMx_1 )
      I_Contact( #pHsMx_2 )
      I_Contact( #EstadoZona.PerReset_CBx )
      Contact( #EstadoZona.Marcha_CBx )
      I_Contact( #Selec_M1_Salida )
      I_Contact( #Selec_M3_Salida )
      I_Contact( #Selec_M1_Entrada )
      I_Contact( #Selec_M3_Entrada )
      wire#w1
      S_SR(operand := #Mx_ET01, r1 := wire#w2)
   END_RUNG
   RUNG wire#powerrail
      Contact( #Mx_ET51 )
      Contact( #Mx_ET151 )
      I_Contact( #Simultaneo_Mx )
      I_Contact( #EstadoVI.Descarga_Act )
   END_RUNG wire#w1
   RUNG wire#powerrail
      Contact( #Mx_ET10 )
      Contact( #Mx_ET110 )
   END_RUNG wire#w2
   // the same network as SCL:
   IF (#Mx_ET00 AND NOT #pHsMx_1 AND NOT #pHsMx_2 AND NOT #EstadoZona.PerReset_CBx AND #EstadoZona.Marcha_CBx AND NOT #Selec_M1_Salida AND NOT #Selec_M3_Salida AND NOT #Selec_M1_Entrada AND NOT #Selec_M3_Entrada) OR (#Mx_ET51 AND #Mx_ET151 AND NOT #Simultaneo_Mx AND NOT #EstadoVI.Descarga_Act) THEN
       #Mx_ET01 := TRUE;   // SR flip-flop
   END_IF;
   IF #Mx_ET10 AND #Mx_ET110 THEN #Mx_ET01 := FALSE; END_IF;
END_REGION

REGION Network 30: ET00 - ESTADO DE INICIO
   RUNG wire#powerrail
      I_Contact( #Mx_ET10 )
      I_Contact( #Mx_ET11 )
      I_Contact( #Mx_ET12 )
      I_Contact( #Mx_ET13 )
      I_Contact( #Mx_ET110 )
      I_Contact( #Mx_ET111 )
      Coil( #Aux_ET00 )
   END_RUNG
   // the same network as SCL:
   #Aux_ET00 := NOT #Mx_ET10 AND NOT #Mx_ET11 AND NOT #Mx_ET12 AND NOT #Mx_ET13 AND NOT #Mx_ET110 AND NOT #Mx_ET111;
END_REGION

REGION Network 31: ----
   RUNG wire#powerrail
      Contact( #Aux_ET00 )
      I_Contact( #Mx_ET50 )
      I_Contact( #Mx_ET51 )
      I_Contact( #Mx_ET150 )
      I_Contact( #Mx_ET151 )
      Coil( #Aux_ET00 )
   END_RUNG
   // the same network as SCL:
   #Aux_ET00 := #Aux_ET00 AND NOT #Mx_ET50 AND NOT #Mx_ET51 AND NOT #Mx_ET150 AND NOT #Mx_ET151;
END_REGION

REGION Network 32: ----
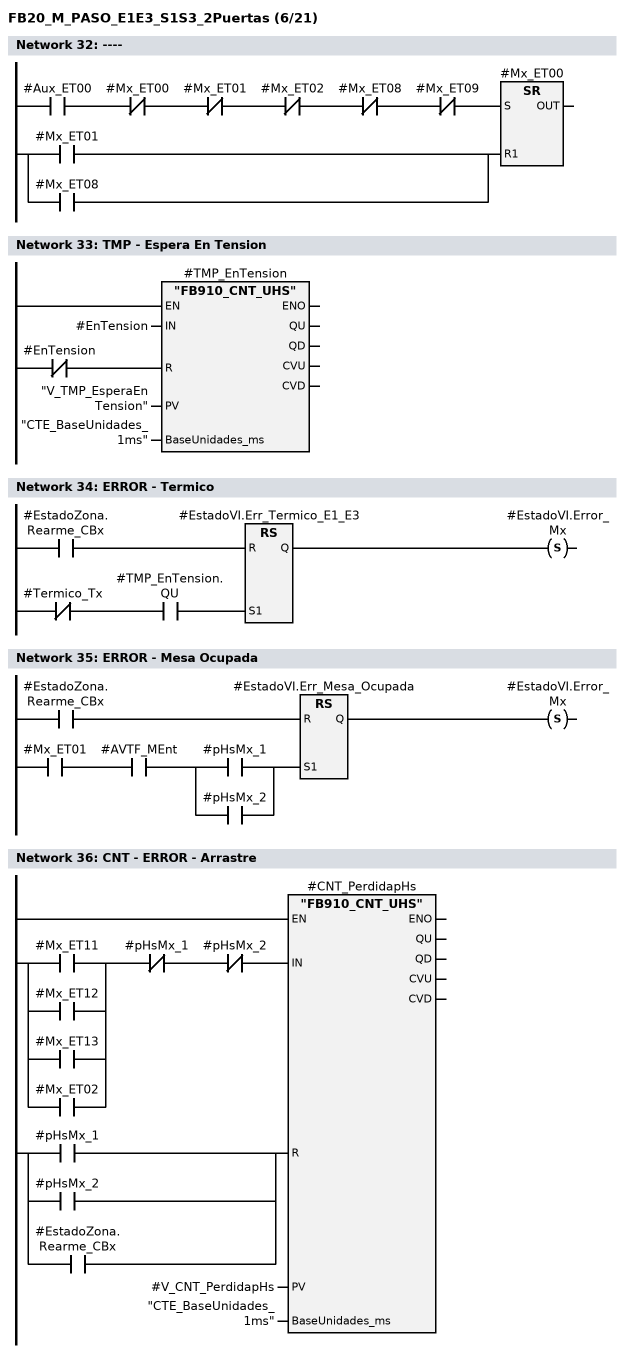
   RUNG wire#powerrail
      Contact( #Aux_ET00 )
      I_Contact( #Mx_ET00 )
      I_Contact( #Mx_ET01 )
      I_Contact( #Mx_ET02 )
      I_Contact( #Mx_ET08 )
      I_Contact( #Mx_ET09 )
      S_SR(operand := #Mx_ET00, r1 := wire#w1)
   END_RUNG
   RUNG wire#powerrail
      Contact( #Mx_ET01 )
   END_RUNG wire#w1
   RUNG wire#powerrail
      Contact( #Mx_ET08 )
   END_RUNG wire#w1
   // the same network as SCL:
   IF #Aux_ET00 AND NOT #Mx_ET00 AND NOT #Mx_ET01 AND NOT #Mx_ET02 AND NOT #Mx_ET08 AND NOT #Mx_ET09 THEN
       #Mx_ET00 := TRUE;   // SR flip-flop
   END_IF;
   IF #Mx_ET01 OR #Mx_ET08 THEN #Mx_ET00 := FALSE; END_IF;
END_REGION

REGION Network 33: TMP - Espera En Tension
   RUNG wire#powerrail
      #TMP_EnTension(R := wire#w1, IN := #EnTension, PV := "V_TMP_EsperaEnTension", BaseUnidades_ms := "CTE_BaseUnidades_1ms", QU =>, QD =>, CVU =>, CVD =>)
   END_RUNG
   RUNG wire#powerrail
      I_Contact( #EnTension )
   END_RUNG wire#w1
   // the same network as SCL:
   #TMP_EnTension(IN := #EnTension,   // "FB910_CNT_UHS"
                  R := NOT #EnTension,
                  PV := "V_TMP_EsperaEnTension",
                  BaseUnidades_ms := "CTE_BaseUnidades_1ms");
END_REGION

REGION Network 34: ERROR - Termico
   RUNG wire#powerrail
      Contact( #EstadoZona.Rearme_CBx )
      S_RS(operand := #EstadoVI.Err_Termico_E1_E3, s1 := wire#w1)
      S_Coil( #EstadoVI.Error_Mx )
   END_RUNG
   RUNG wire#powerrail
      I_Contact( #Termico_Tx )
      Contact( #TMP_EnTension.QU )
   END_RUNG wire#w1
   // the same network as SCL:
   IF #EstadoZona.Rearme_CBx THEN
       #EstadoVI.Err_Termico_E1_E3 := FALSE;   // RS flip-flop
   END_IF;
   IF NOT #Termico_Tx AND #TMP_EnTension.QU THEN #EstadoVI.Err_Termico_E1_E3 := TRUE; END_IF;
   IF #EstadoVI.Err_Termico_E1_E3 THEN #EstadoVI.Error_Mx := TRUE; END_IF;
END_REGION

REGION Network 35: ERROR - Mesa Ocupada
   RUNG wire#powerrail
      Contact( #EstadoZona.Rearme_CBx )
      S_RS(operand := #EstadoVI.Err_Mesa_Ocupada, s1 := wire#w2)
      S_Coil( #EstadoVI.Error_Mx )
   END_RUNG
   RUNG wire#powerrail
      Contact( #Mx_ET01 )
      Contact( #AVTF_MEnt )
      wire#w1
      Contact( #pHsMx_1 )
   END_RUNG wire#w2
   RUNG wire#w1
      Contact( #pHsMx_2 )
   END_RUNG wire#w2
   // the same network as SCL:
   IF #EstadoZona.Rearme_CBx THEN
       #EstadoVI.Err_Mesa_Ocupada := FALSE;   // RS flip-flop
   END_IF;
   IF #Mx_ET01 AND #AVTF_MEnt AND (#pHsMx_1 OR #pHsMx_2) THEN #EstadoVI.Err_Mesa_Ocupada := TRUE; END_IF;
   IF #EstadoVI.Err_Mesa_Ocupada THEN #EstadoVI.Error_Mx := TRUE; END_IF;
END_REGION

REGION Network 36: CNT - ERROR - Arrastre
   RUNG wire#powerrail
      #CNT_PerdidapHs(IN := wire#w2, R := wire#w3, PV := #V_CNT_PerdidapHs, BaseUnidades_ms := "CTE_BaseUnidades_1ms", QU =>, QD =>, CVU =>, CVD =>)
   END_RUNG
   RUNG wire#powerrail
      Contact( #Mx_ET11 )
      wire#w1
      I_Contact( #pHsMx_1 )
      I_Contact( #pHsMx_2 )
   END_RUNG wire#w2
   RUNG wire#powerrail
      Contact( #Mx_ET12 )
   END_RUNG wire#w1
   RUNG wire#powerrail
      Contact( #Mx_ET13 )
   END_RUNG wire#w1
   RUNG wire#powerrail
      Contact( #Mx_ET02 )
   END_RUNG wire#w1
   RUNG wire#powerrail
      Contact( #pHsMx_1 )
   END_RUNG wire#w3
   RUNG wire#powerrail
      Contact( #pHsMx_2 )
   END_RUNG wire#w3
   RUNG wire#powerrail
      Contact( #EstadoZona.Rearme_CBx )
   END_RUNG wire#w3
   // the same network as SCL:
   #CNT_PerdidapHs(IN := (#Mx_ET11 OR #Mx_ET12 OR #Mx_ET13 OR #Mx_ET02) AND NOT #pHsMx_1 AND NOT #pHsMx_2,   // "FB910_CNT_UHS"
                   R := #pHsMx_1 OR #pHsMx_2 OR #EstadoZona.Rearme_CBx,
                   PV := #V_CNT_PerdidapHs,
                   BaseUnidades_ms := "CTE_BaseUnidades_1ms");
END_REGION

REGION Network 37: ERROR - Arrastre
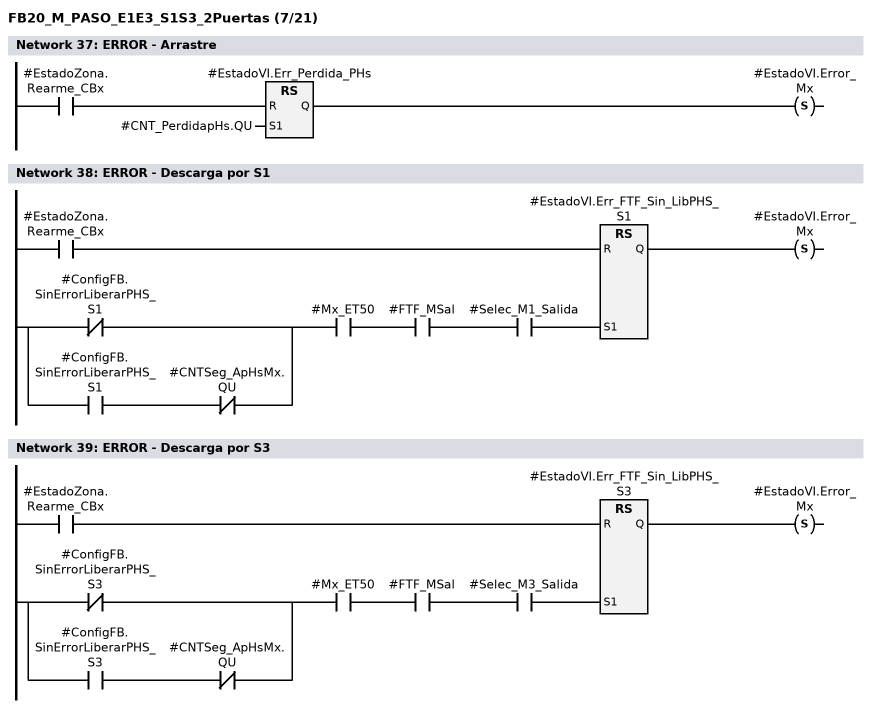
   RUNG wire#powerrail
      Contact( #EstadoZona.Rearme_CBx )
      S_RS(operand := #EstadoVI.Err_Perdida_PHs, s1 := #CNT_PerdidapHs.QU)
      S_Coil( #EstadoVI.Error_Mx )
   END_RUNG
   // the same network as SCL:
   IF #EstadoZona.Rearme_CBx THEN
       #EstadoVI.Err_Perdida_PHs := FALSE;   // RS flip-flop
   END_IF;
   IF #CNT_PerdidapHs.QU THEN #EstadoVI.Err_Perdida_PHs := TRUE; END_IF;
   IF #EstadoVI.Err_Perdida_PHs THEN #EstadoVI.Error_Mx := TRUE; END_IF;
END_REGION

REGION Network 38: ERROR - Descarga por S1
   RUNG wire#powerrail
      Contact( #EstadoZona.Rearme_CBx )
      S_RS(operand := #EstadoVI.Err_FTF_Sin_LibPHS_S1, s1 := wire#w2)
      S_Coil( #EstadoVI.Error_Mx )
   END_RUNG
   RUNG wire#powerrail
      I_Contact( #ConfigFB.SinErrorLiberarPHS_S1 )
      wire#w1
      Contact( #Mx_ET50 )
      Contact( #FTF_MSal )
      Contact( #Selec_M1_Salida )
   END_RUNG wire#w2
   RUNG wire#powerrail
      Contact( #ConfigFB.SinErrorLiberarPHS_S1 )
      I_Contact( #CNTSeg_ApHsMx.QU )
   END_RUNG wire#w1
   // the same network as SCL:
   IF #EstadoZona.Rearme_CBx THEN
       #EstadoVI.Err_FTF_Sin_LibPHS_S1 := FALSE;   // RS flip-flop
   END_IF;
   IF (NOT #ConfigFB.SinErrorLiberarPHS_S1 OR (#ConfigFB.SinErrorLiberarPHS_S1 AND NOT #CNTSeg_ApHsMx.QU)) AND #Mx_ET50 AND #FTF_MSal AND #Selec_M1_Salida THEN
       #EstadoVI.Err_FTF_Sin_LibPHS_S1 := TRUE;
   END_IF;
   IF #EstadoVI.Err_FTF_Sin_LibPHS_S1 THEN #EstadoVI.Error_Mx := TRUE; END_IF;
END_REGION

REGION Network 39: ERROR - Descarga por S3
   RUNG wire#powerrail
      Contact( #EstadoZona.Rearme_CBx )
      S_RS(operand := #EstadoVI.Err_FTF_Sin_LibPHS_S3, s1 := wire#w2)
      S_Coil( #EstadoVI.Error_Mx )
   END_RUNG
   RUNG wire#powerrail
      I_Contact( #ConfigFB.SinErrorLiberarPHS_S3 )
      wire#w1
      Contact( #Mx_ET50 )
      Contact( #FTF_MSal )
      Contact( #Selec_M3_Salida )
   END_RUNG wire#w2
   RUNG wire#powerrail
      Contact( #ConfigFB.SinErrorLiberarPHS_S3 )
      I_Contact( #CNTSeg_ApHsMx.QU )
   END_RUNG wire#w1
   // the same network as SCL:
   IF #EstadoZona.Rearme_CBx THEN
       #EstadoVI.Err_FTF_Sin_LibPHS_S3 := FALSE;   // RS flip-flop
   END_IF;
   IF (NOT #ConfigFB.SinErrorLiberarPHS_S3 OR (#ConfigFB.SinErrorLiberarPHS_S3 AND NOT #CNTSeg_ApHsMx.QU)) AND #Mx_ET50 AND #FTF_MSal AND #Selec_M3_Salida THEN
       #EstadoVI.Err_FTF_Sin_LibPHS_S3 := TRUE;
   END_IF;
   IF #EstadoVI.Err_FTF_Sin_LibPHS_S3 THEN #EstadoVI.Error_Mx := TRUE; END_IF;
END_REGION

REGION Network 40: TMP - ERROR - TimeOut Avance
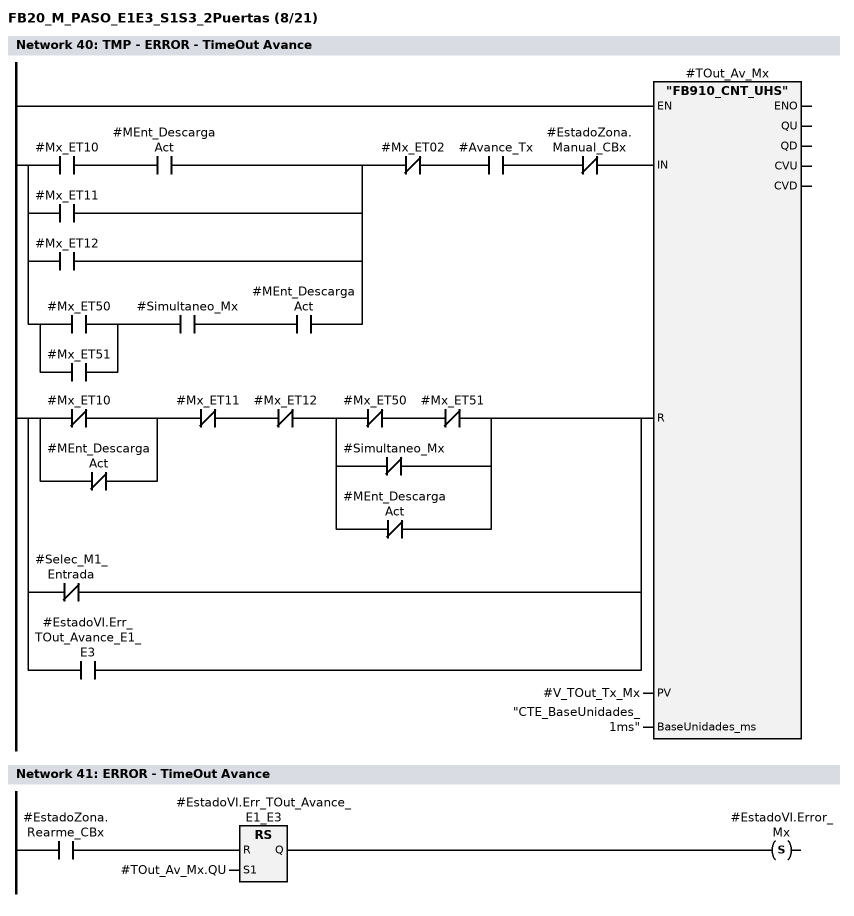
   RUNG wire#powerrail
      #TOut_Av_Mx(IN := wire#w3, R := wire#w6, PV := #V_TOut_Tx_Mx, BaseUnidades_ms := "CTE_BaseUnidades_1ms", QU =>, QD =>, CVU =>, CVD =>)
   END_RUNG
   RUNG wire#powerrail
      Contact( #Mx_ET10 )
      Contact( #MEnt_DescargaAct )
      wire#w1
      I_Contact( #Mx_ET02 )
      Contact( #Avance_Tx )
      I_Contact( #EstadoZona.Manual_CBx )
   END_RUNG wire#w3
   RUNG wire#powerrail
      Contact( #Mx_ET11 )
   END_RUNG wire#w1
   RUNG wire#powerrail
      Contact( #Mx_ET12 )
   END_RUNG wire#w1
   RUNG wire#powerrail
      Contact( #Mx_ET50 )
      wire#w2
      Contact( #Simultaneo_Mx )
      Contact( #MEnt_DescargaAct )
   END_RUNG wire#w1
   RUNG wire#powerrail
      Contact( #Mx_ET51 )
   END_RUNG wire#w2
   RUNG wire#powerrail
      I_Contact( #Mx_ET10 )
      wire#w4
      I_Contact( #Mx_ET11 )
      I_Contact( #Mx_ET12 )
      wire#w5
      I_Contact( #Mx_ET50 )
      I_Contact( #Mx_ET51 )
   END_RUNG wire#w6
   RUNG wire#powerrail
      I_Contact( #MEnt_DescargaAct )
   END_RUNG wire#w4
   RUNG wire#w5
      I_Contact( #Simultaneo_Mx )
   END_RUNG wire#w6
   RUNG wire#w5
      I_Contact( #MEnt_DescargaAct )
   END_RUNG wire#w6
   RUNG wire#powerrail
      I_Contact( #Selec_M1_Entrada )
   END_RUNG wire#w6
   RUNG wire#powerrail
      Contact( #EstadoVI.Err_TOut_Avance_E1_E3 )
   END_RUNG wire#w6
   // the same network as SCL:
   #TOut_Av_Mx(IN := ((#Mx_ET10 AND #MEnt_DescargaAct) OR #Mx_ET11 OR #Mx_ET12 OR ((#Mx_ET50 OR #Mx_ET51) AND #Simultaneo_Mx AND #MEnt_DescargaAct)) AND NOT #Mx_ET02 AND #Avance_Tx AND NOT #EstadoZona.Manual_CBx,   // "FB910_CNT_UHS"
               R := ((NOT #Mx_ET10 OR NOT #MEnt_DescargaAct) AND NOT #Mx_ET11 AND NOT #Mx_ET12 AND ((NOT #Mx_ET50 AND NOT #Mx_ET51) OR NOT #Simultaneo_Mx OR NOT #MEnt_DescargaAct)) OR NOT #Selec_M1_Entrada OR #EstadoVI.Err_TOut_Avance_E1_E3,
               PV := #V_TOut_Tx_Mx,
               BaseUnidades_ms := "CTE_BaseUnidades_1ms");
END_REGION

REGION Network 41: ERROR - TimeOut Avance
   RUNG wire#powerrail
      Contact( #EstadoZona.Rearme_CBx )
      S_RS(operand := #EstadoVI.Err_TOut_Avance_E1_E3, s1 := #TOut_Av_Mx.QU)
      S_Coil( #EstadoVI.Error_Mx )
   END_RUNG
   // the same network as SCL:
   IF #EstadoZona.Rearme_CBx THEN
       #EstadoVI.Err_TOut_Avance_E1_E3 := FALSE;   // RS flip-flop
   END_IF;
   IF #TOut_Av_Mx.QU THEN #EstadoVI.Err_TOut_Avance_E1_E3 := TRUE; END_IF;
   IF #EstadoVI.Err_TOut_Avance_E1_E3 THEN #EstadoVI.Error_Mx := TRUE; END_IF;
END_REGION

REGION Network 42: TMP - ERROR - TimeOut Retroceso
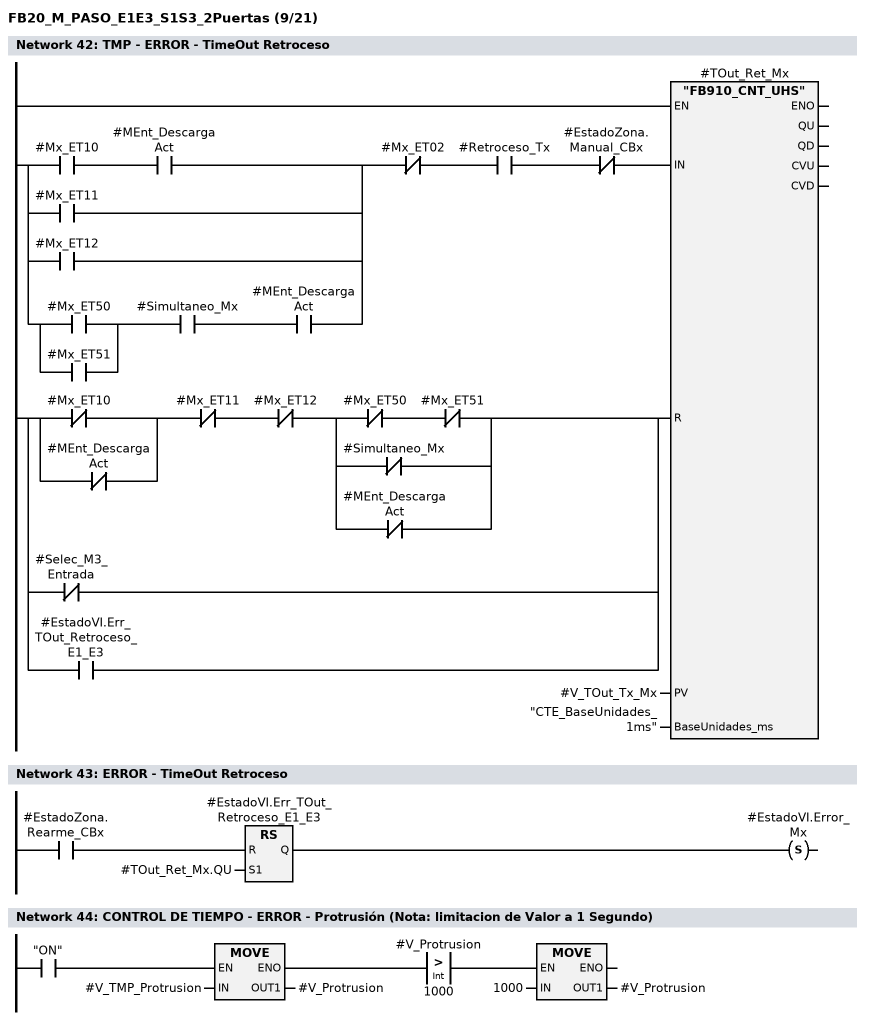
   RUNG wire#powerrail
      #TOut_Ret_Mx(IN := wire#w3, R := wire#w6, PV := #V_TOut_Tx_Mx, BaseUnidades_ms := "CTE_BaseUnidades_1ms", QU =>, QD =>, CVU =>, CVD =>)
   END_RUNG
   RUNG wire#powerrail
      Contact( #Mx_ET10 )
      Contact( #MEnt_DescargaAct )
      wire#w1
      I_Contact( #Mx_ET02 )
      Contact( #Retroceso_Tx )
      I_Contact( #EstadoZona.Manual_CBx )
   END_RUNG wire#w3
   RUNG wire#powerrail
      Contact( #Mx_ET11 )
   END_RUNG wire#w1
   RUNG wire#powerrail
      Contact( #Mx_ET12 )
   END_RUNG wire#w1
   RUNG wire#powerrail
      Contact( #Mx_ET50 )
      wire#w2
      Contact( #Simultaneo_Mx )
      Contact( #MEnt_DescargaAct )
   END_RUNG wire#w1
   RUNG wire#powerrail
      Contact( #Mx_ET51 )
   END_RUNG wire#w2
   RUNG wire#powerrail
      I_Contact( #Mx_ET10 )
      wire#w4
      I_Contact( #Mx_ET11 )
      I_Contact( #Mx_ET12 )
      wire#w5
      I_Contact( #Mx_ET50 )
      I_Contact( #Mx_ET51 )
   END_RUNG wire#w6
   RUNG wire#powerrail
      I_Contact( #MEnt_DescargaAct )
   END_RUNG wire#w4
   RUNG wire#w5
      I_Contact( #Simultaneo_Mx )
   END_RUNG wire#w6
   RUNG wire#w5
      I_Contact( #MEnt_DescargaAct )
   END_RUNG wire#w6
   RUNG wire#powerrail
      I_Contact( #Selec_M3_Entrada )
   END_RUNG wire#w6
   RUNG wire#powerrail
      Contact( #EstadoVI.Err_TOut_Retroceso_E1_E3 )
   END_RUNG wire#w6
   // the same network as SCL:
   #TOut_Ret_Mx(IN := ((#Mx_ET10 AND #MEnt_DescargaAct) OR #Mx_ET11 OR #Mx_ET12 OR ((#Mx_ET50 OR #Mx_ET51) AND #Simultaneo_Mx AND #MEnt_DescargaAct)) AND NOT #Mx_ET02 AND #Retroceso_Tx AND NOT #EstadoZona.Manual_CBx,   // "FB910_CNT_UHS"
                R := ((NOT #Mx_ET10 OR NOT #MEnt_DescargaAct) AND NOT #Mx_ET11 AND NOT #Mx_ET12 AND ((NOT #Mx_ET50 AND NOT #Mx_ET51) OR NOT #Simultaneo_Mx OR NOT #MEnt_DescargaAct)) OR NOT #Selec_M3_Entrada OR #EstadoVI.Err_TOut_Retroceso_E1_E3,
                PV := #V_TOut_Tx_Mx,
                BaseUnidades_ms := "CTE_BaseUnidades_1ms");
END_REGION

REGION Network 43: ERROR - TimeOut Retroceso
   RUNG wire#powerrail
      Contact( #EstadoZona.Rearme_CBx )
      S_RS(operand := #EstadoVI.Err_TOut_Retroceso_E1_E3, s1 := #TOut_Ret_Mx.QU)
      S_Coil( #EstadoVI.Error_Mx )
   END_RUNG
   // the same network as SCL:
   IF #EstadoZona.Rearme_CBx THEN
       #EstadoVI.Err_TOut_Retroceso_E1_E3 := FALSE;   // RS flip-flop
   END_IF;
   IF #TOut_Ret_Mx.QU THEN #EstadoVI.Err_TOut_Retroceso_E1_E3 := TRUE; END_IF;
   IF #EstadoVI.Err_TOut_Retroceso_E1_E3 THEN #EstadoVI.Error_Mx := TRUE; END_IF;
END_REGION

REGION Network 44: CONTROL DE TIEMPO - ERROR - Protrusión (Nota: limitacion de Valor a 1 Segundo)
   RUNG wire#powerrail
      Contact( "ON" )
      Move(in := #V_TMP_Protrusion, out1 => #V_Protrusion)
      { S7_Templates := "SrcType := Int" } GT_Contact(in1 := #V_Protrusion, in2 := 1000)
      Move(in := 1000, out1 => #V_Protrusion)
   END_RUNG
   // the same network as SCL:
   IF "ON" THEN #V_Protrusion := #V_TMP_Protrusion; END_IF;
   IF "ON" AND (#V_Protrusion > 1000) THEN #V_Protrusion := 1000; END_IF;
END_REGION

REGION Network 45: TMP - ERROR - Protrusión
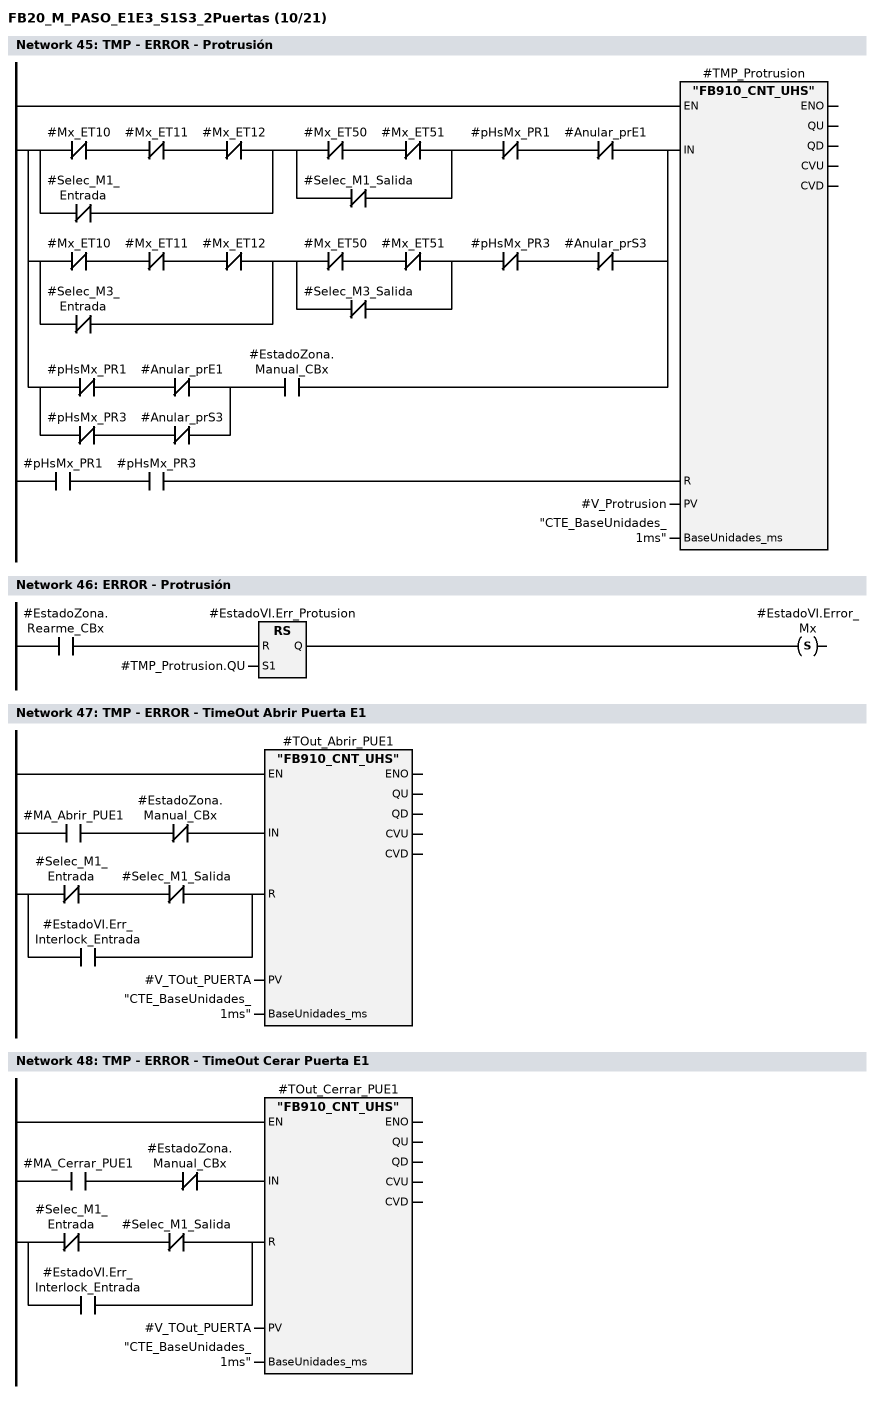
   RUNG wire#powerrail
      #TMP_Protrusion(IN := wire#w6, R := wire#w7, PV := #V_Protrusion, BaseUnidades_ms := "CTE_BaseUnidades_1ms", QU =>, QD =>, CVU =>, CVD =>)
   END_RUNG
   RUNG wire#powerrail
      I_Contact( #Mx_ET10 )
      I_Contact( #Mx_ET11 )
      I_Contact( #Mx_ET12 )
      wire#w1
      I_Contact( #Mx_ET50 )
      I_Contact( #Mx_ET51 )
      wire#w2
      I_Contact( #pHsMx_PR1 )
      I_Contact( #Anular_prE1 )
   END_RUNG wire#w6
   RUNG wire#powerrail
      I_Contact( #Selec_M1_Entrada )
   END_RUNG wire#w1
   RUNG wire#w1
      I_Contact( #Selec_M1_Salida )
   END_RUNG wire#w2
   RUNG wire#powerrail
      I_Contact( #Mx_ET10 )
      I_Contact( #Mx_ET11 )
      I_Contact( #Mx_ET12 )
      wire#w3
      I_Contact( #Mx_ET50 )
      I_Contact( #Mx_ET51 )
      wire#w4
      I_Contact( #pHsMx_PR3 )
      I_Contact( #Anular_prS3 )
   END_RUNG wire#w6
   RUNG wire#powerrail
      I_Contact( #Selec_M3_Entrada )
   END_RUNG wire#w3
   RUNG wire#w3
      I_Contact( #Selec_M3_Salida )
   END_RUNG wire#w4
   RUNG wire#powerrail
      I_Contact( #pHsMx_PR1 )
      I_Contact( #Anular_prE1 )
      wire#w5
      Contact( #EstadoZona.Manual_CBx )
   END_RUNG wire#w6
   RUNG wire#powerrail
      I_Contact( #pHsMx_PR3 )
      I_Contact( #Anular_prS3 )
   END_RUNG wire#w5
   RUNG wire#powerrail
      Contact( #pHsMx_PR1 )
      Contact( #pHsMx_PR3 )
   END_RUNG wire#w7
   // the same network as SCL:
   #TMP_Protrusion(IN := (((NOT #Mx_ET10 AND NOT #Mx_ET11 AND NOT #Mx_ET12) OR NOT #Selec_M1_Entrada) AND ((NOT #Mx_ET50 AND NOT #Mx_ET51) OR NOT #Selec_M1_Salida) AND NOT #pHsMx_PR1 AND NOT #Anular_prE1) OR (((NOT #Mx_ET10 AND NOT #Mx_ET11 AND NOT #Mx_ET12) OR NOT #Selec_M3_Entrada) AND ((NOT #Mx_ET50 AND NOT #Mx_ET51) OR NOT #Selec_M3_Salida) AND NOT #pHsMx_PR3 AND NOT #Anular_prS3) OR (((NOT #pHsMx_PR1 AND NOT #Anular_prE1) OR (NOT #pHsMx_PR3 AND NOT #Anular_prS3)) AND #EstadoZona.Manual_CBx),   // "FB910_CNT_UHS"
                   R := #pHsMx_PR1 AND #pHsMx_PR3,
                   PV := #V_Protrusion,
                   BaseUnidades_ms := "CTE_BaseUnidades_1ms");
END_REGION

REGION Network 46: ERROR - Protrusión
   RUNG wire#powerrail
      Contact( #EstadoZona.Rearme_CBx )
      S_RS(operand := #EstadoVI.Err_Protusion, s1 := #TMP_Protrusion.QU)
      S_Coil( #EstadoVI.Error_Mx )
   END_RUNG
   // the same network as SCL:
   IF #EstadoZona.Rearme_CBx THEN
       #EstadoVI.Err_Protusion := FALSE;   // RS flip-flop
   END_IF;
   IF #TMP_Protrusion.QU THEN #EstadoVI.Err_Protusion := TRUE; END_IF;
   IF #EstadoVI.Err_Protusion THEN #EstadoVI.Error_Mx := TRUE; END_IF;
END_REGION

REGION Network 47: TMP - ERROR - TimeOut Abrir Puerta E1
   RUNG wire#powerrail
      #TOut_Abrir_PUE1(IN := wire#w1, R := wire#w2, PV := #V_TOut_PUERTA, BaseUnidades_ms := "CTE_BaseUnidades_1ms", QU =>, QD =>, CVU =>, CVD =>)
   END_RUNG
   RUNG wire#powerrail
      Contact( #MA_Abrir_PUE1 )
      I_Contact( #EstadoZona.Manual_CBx )
   END_RUNG wire#w1
   RUNG wire#powerrail
      I_Contact( #Selec_M1_Entrada )
      I_Contact( #Selec_M1_Salida )
   END_RUNG wire#w2
   RUNG wire#powerrail
      Contact( #EstadoVI.Err_Interlock_Entrada )
   END_RUNG wire#w2
   // the same network as SCL:
   #TOut_Abrir_PUE1(IN := #MA_Abrir_PUE1 AND NOT #EstadoZona.Manual_CBx,   // "FB910_CNT_UHS"
                    R := (NOT #Selec_M1_Entrada AND NOT #Selec_M1_Salida) OR #EstadoVI.Err_Interlock_Entrada,
                    PV := #V_TOut_PUERTA,
                    BaseUnidades_ms := "CTE_BaseUnidades_1ms");
END_REGION

REGION Network 48: TMP - ERROR - TimeOut Cerar Puerta E1
   RUNG wire#powerrail
      #TOut_Cerrar_PUE1(IN := wire#w1, R := wire#w2, PV := #V_TOut_PUERTA, BaseUnidades_ms := "CTE_BaseUnidades_1ms", QU =>, QD =>, CVU =>, CVD =>)
   END_RUNG
   RUNG wire#powerrail
      Contact( #MA_Cerrar_PUE1 )
      I_Contact( #EstadoZona.Manual_CBx )
   END_RUNG wire#w1
   RUNG wire#powerrail
      I_Contact( #Selec_M1_Entrada )
      I_Contact( #Selec_M1_Salida )
   END_RUNG wire#w2
   RUNG wire#powerrail
      Contact( #EstadoVI.Err_Interlock_Entrada )
   END_RUNG wire#w2
   // the same network as SCL:
   #TOut_Cerrar_PUE1(IN := #MA_Cerrar_PUE1 AND NOT #EstadoZona.Manual_CBx,   // "FB910_CNT_UHS"
                     R := (NOT #Selec_M1_Entrada AND NOT #Selec_M1_Salida) OR #EstadoVI.Err_Interlock_Entrada,
                     PV := #V_TOut_PUERTA,
                     BaseUnidades_ms := "CTE_BaseUnidades_1ms");
END_REGION

REGION Network 49: ERROR - Movimiento de la Puerta E1
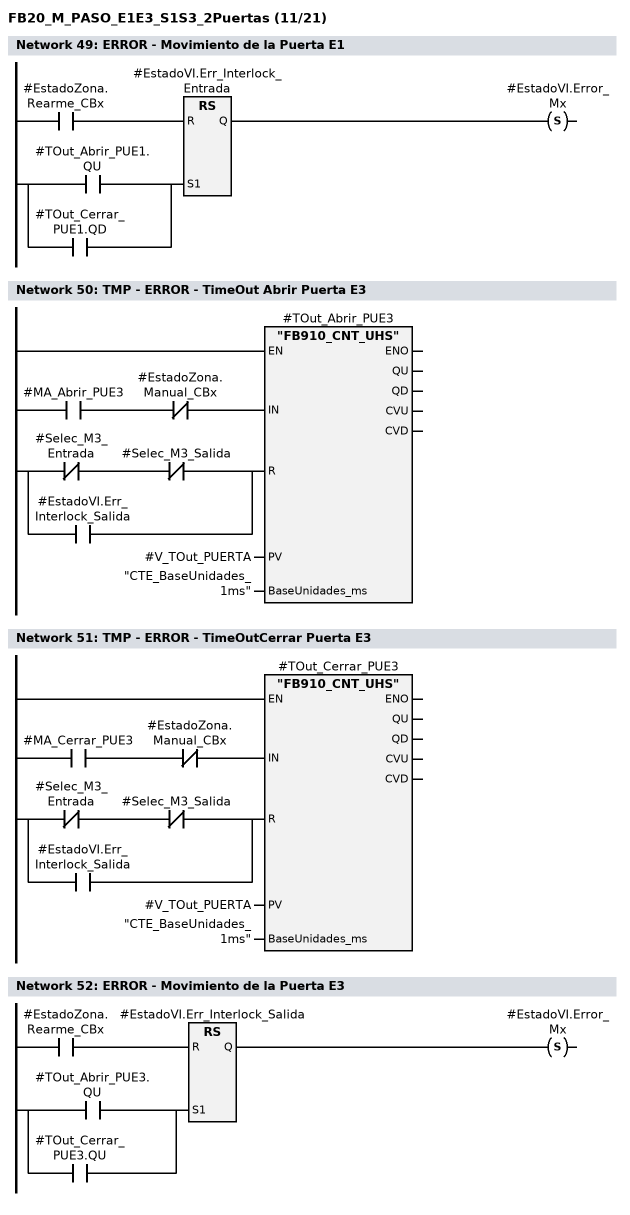
   RUNG wire#powerrail
      Contact( #EstadoZona.Rearme_CBx )
      S_RS(operand := #EstadoVI.Err_Interlock_Entrada, s1 := wire#w1)
      S_Coil( #EstadoVI.Error_Mx )
   END_RUNG
   RUNG wire#powerrail
      Contact( #TOut_Abrir_PUE1.QU )
   END_RUNG wire#w1
   RUNG wire#powerrail
      Contact( #TOut_Cerrar_PUE1.QD )
   END_RUNG wire#w1
   // the same network as SCL:
   IF #EstadoZona.Rearme_CBx THEN
       #EstadoVI.Err_Interlock_Entrada := FALSE;   // RS flip-flop
   END_IF;
   IF #TOut_Abrir_PUE1.QU OR #TOut_Cerrar_PUE1.QD THEN #EstadoVI.Err_Interlock_Entrada := TRUE; END_IF;
   IF #EstadoVI.Err_Interlock_Entrada THEN #EstadoVI.Error_Mx := TRUE; END_IF;
END_REGION

REGION Network 50: TMP - ERROR - TimeOut Abrir Puerta E3
   RUNG wire#powerrail
      #TOut_Abrir_PUE3(IN := wire#w1, R := wire#w2, PV := #V_TOut_PUERTA, BaseUnidades_ms := "CTE_BaseUnidades_1ms", QU =>, QD =>, CVU =>, CVD =>)
   END_RUNG
   RUNG wire#powerrail
      Contact( #MA_Abrir_PUE3 )
      I_Contact( #EstadoZona.Manual_CBx )
   END_RUNG wire#w1
   RUNG wire#powerrail
      I_Contact( #Selec_M3_Entrada )
      I_Contact( #Selec_M3_Salida )
   END_RUNG wire#w2
   RUNG wire#powerrail
      Contact( #EstadoVI.Err_Interlock_Salida )
   END_RUNG wire#w2
   // the same network as SCL:
   #TOut_Abrir_PUE3(IN := #MA_Abrir_PUE3 AND NOT #EstadoZona.Manual_CBx,   // "FB910_CNT_UHS"
                    R := (NOT #Selec_M3_Entrada AND NOT #Selec_M3_Salida) OR #EstadoVI.Err_Interlock_Salida,
                    PV := #V_TOut_PUERTA,
                    BaseUnidades_ms := "CTE_BaseUnidades_1ms");
END_REGION

REGION Network 51: TMP - ERROR - TimeOutCerrar Puerta E3
   RUNG wire#powerrail
      #TOut_Cerrar_PUE3(IN := wire#w1, R := wire#w2, PV := #V_TOut_PUERTA, BaseUnidades_ms := "CTE_BaseUnidades_1ms", QU =>, QD =>, CVU =>, CVD =>)
   END_RUNG
   RUNG wire#powerrail
      Contact( #MA_Cerrar_PUE3 )
      I_Contact( #EstadoZona.Manual_CBx )
   END_RUNG wire#w1
   RUNG wire#powerrail
      I_Contact( #Selec_M3_Entrada )
      I_Contact( #Selec_M3_Salida )
   END_RUNG wire#w2
   RUNG wire#powerrail
      Contact( #EstadoVI.Err_Interlock_Salida )
   END_RUNG wire#w2
   // the same network as SCL:
   #TOut_Cerrar_PUE3(IN := #MA_Cerrar_PUE3 AND NOT #EstadoZona.Manual_CBx,   // "FB910_CNT_UHS"
                     R := (NOT #Selec_M3_Entrada AND NOT #Selec_M3_Salida) OR #EstadoVI.Err_Interlock_Salida,
                     PV := #V_TOut_PUERTA,
                     BaseUnidades_ms := "CTE_BaseUnidades_1ms");
END_REGION

REGION Network 52: ERROR - Movimiento de la Puerta E3
   RUNG wire#powerrail
      Contact( #EstadoZona.Rearme_CBx )
      S_RS(operand := #EstadoVI.Err_Interlock_Salida, s1 := wire#w1)
      S_Coil( #EstadoVI.Error_Mx )
   END_RUNG
   RUNG wire#powerrail
      Contact( #TOut_Abrir_PUE3.QU )
   END_RUNG wire#w1
   RUNG wire#powerrail
      Contact( #TOut_Cerrar_PUE3.QU )
   END_RUNG wire#w1
   // the same network as SCL:
   IF #EstadoZona.Rearme_CBx THEN
       #EstadoVI.Err_Interlock_Salida := FALSE;   // RS flip-flop
   END_IF;
   IF #TOut_Abrir_PUE3.QU OR #TOut_Cerrar_PUE3.QU THEN #EstadoVI.Err_Interlock_Salida := TRUE; END_IF;
   IF #EstadoVI.Err_Interlock_Salida THEN #EstadoVI.Error_Mx := TRUE; END_IF;
END_REGION

REGION Network 53: ERROR - Abertura de Puertas
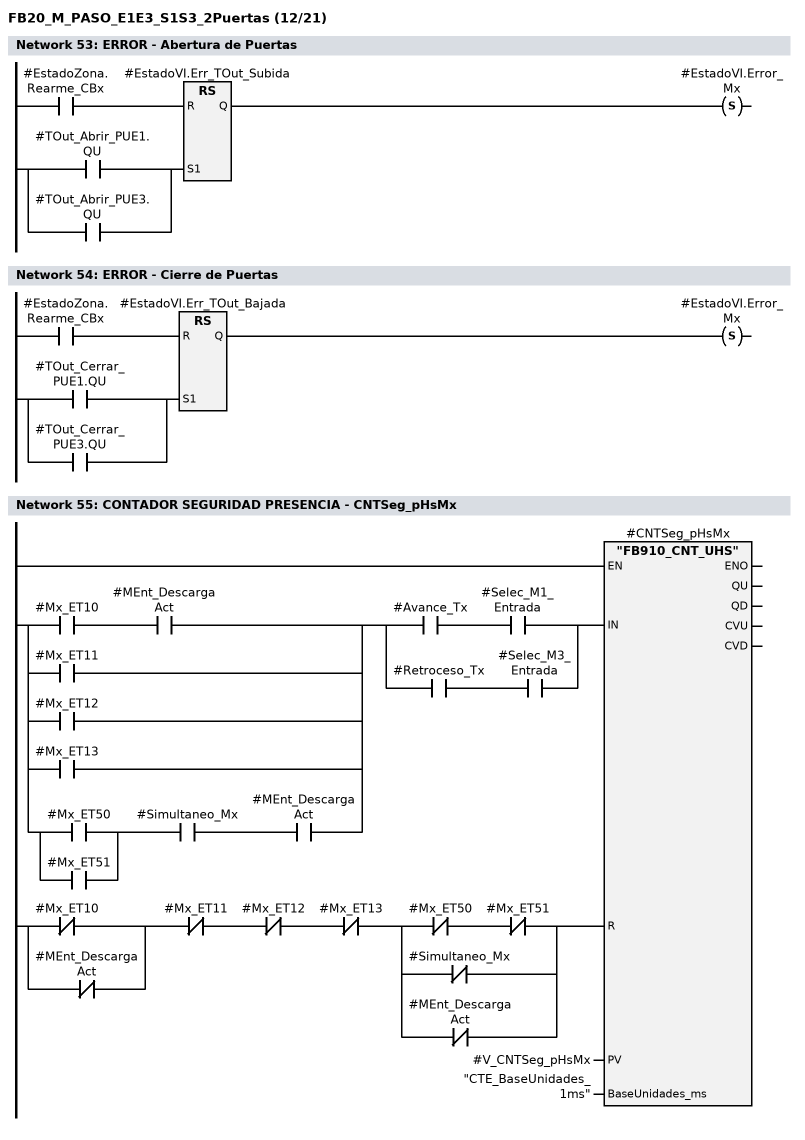
   RUNG wire#powerrail
      Contact( #EstadoZona.Rearme_CBx )
      S_RS(operand := #EstadoVI.Err_TOut_Subida, s1 := wire#w1)
      S_Coil( #EstadoVI.Error_Mx )
   END_RUNG
   RUNG wire#powerrail
      Contact( #TOut_Abrir_PUE1.QU )
   END_RUNG wire#w1
   RUNG wire#powerrail
      Contact( #TOut_Abrir_PUE3.QU )
   END_RUNG wire#w1
   // the same network as SCL:
   IF #EstadoZona.Rearme_CBx THEN
       #EstadoVI.Err_TOut_Subida := FALSE;   // RS flip-flop
   END_IF;
   IF #TOut_Abrir_PUE1.QU OR #TOut_Abrir_PUE3.QU THEN #EstadoVI.Err_TOut_Subida := TRUE; END_IF;
   IF #EstadoVI.Err_TOut_Subida THEN #EstadoVI.Error_Mx := TRUE; END_IF;
END_REGION

REGION Network 54: ERROR - Cierre de Puertas
   RUNG wire#powerrail
      Contact( #EstadoZona.Rearme_CBx )
      S_RS(operand := #EstadoVI.Err_TOut_Bajada, s1 := wire#w1)
      S_Coil( #EstadoVI.Error_Mx )
   END_RUNG
   RUNG wire#powerrail
      Contact( #TOut_Cerrar_PUE1.QU )
   END_RUNG wire#w1
   RUNG wire#powerrail
      Contact( #TOut_Cerrar_PUE3.QU )
   END_RUNG wire#w1
   // the same network as SCL:
   IF #EstadoZona.Rearme_CBx THEN
       #EstadoVI.Err_TOut_Bajada := FALSE;   // RS flip-flop
   END_IF;
   IF #TOut_Cerrar_PUE1.QU OR #TOut_Cerrar_PUE3.QU THEN #EstadoVI.Err_TOut_Bajada := TRUE; END_IF;
   IF #EstadoVI.Err_TOut_Bajada THEN #EstadoVI.Error_Mx := TRUE; END_IF;
END_REGION

REGION Network 55: CONTADOR SEGURIDAD PRESENCIA - CNTSeg_pHsMx
   RUNG wire#powerrail
      #CNTSeg_pHsMx(IN := wire#w3, R := wire#w6, PV := #V_CNTSeg_pHsMx, BaseUnidades_ms := "CTE_BaseUnidades_1ms", QU =>, QD =>, CVU =>, CVD =>)
   END_RUNG
   RUNG wire#powerrail
      Contact( #Mx_ET10 )
      Contact( #MEnt_DescargaAct )
      wire#w1
      Contact( #Avance_Tx )
      Contact( #Selec_M1_Entrada )
   END_RUNG wire#w3
   RUNG wire#powerrail
      Contact( #Mx_ET11 )
   END_RUNG wire#w1
   RUNG wire#powerrail
      Contact( #Mx_ET12 )
   END_RUNG wire#w1
   RUNG wire#powerrail
      Contact( #Mx_ET13 )
   END_RUNG wire#w1
   RUNG wire#powerrail
      Contact( #Mx_ET50 )
      wire#w2
      Contact( #Simultaneo_Mx )
      Contact( #MEnt_DescargaAct )
   END_RUNG wire#w1
   RUNG wire#powerrail
      Contact( #Mx_ET51 )
   END_RUNG wire#w2
   RUNG wire#w1
      Contact( #Retroceso_Tx )
      Contact( #Selec_M3_Entrada )
   END_RUNG wire#w3
   RUNG wire#powerrail
      I_Contact( #Mx_ET10 )
      wire#w4
      I_Contact( #Mx_ET11 )
      I_Contact( #Mx_ET12 )
      I_Contact( #Mx_ET13 )
      wire#w5
      I_Contact( #Mx_ET50 )
      I_Contact( #Mx_ET51 )
   END_RUNG wire#w6
   RUNG wire#powerrail
      I_Contact( #MEnt_DescargaAct )
   END_RUNG wire#w4
   RUNG wire#w5
      I_Contact( #Simultaneo_Mx )
   END_RUNG wire#w6
   RUNG wire#w5
      I_Contact( #MEnt_DescargaAct )
   END_RUNG wire#w6
   // the same network as SCL:
   #CNTSeg_pHsMx(IN := ((#Mx_ET10 AND #MEnt_DescargaAct) OR #Mx_ET11 OR #Mx_ET12 OR #Mx_ET13 OR ((#Mx_ET50 OR #Mx_ET51) AND #Simultaneo_Mx AND #MEnt_DescargaAct)) AND ((#Avance_Tx AND #Selec_M1_Entrada) OR (#Retroceso_Tx AND #Selec_M3_Entrada)),   // "FB910_CNT_UHS"
                 R := (NOT #Mx_ET10 OR NOT #MEnt_DescargaAct) AND NOT #Mx_ET11 AND NOT #Mx_ET12 AND NOT #Mx_ET13 AND ((NOT #Mx_ET50 AND NOT #Mx_ET51) OR NOT #Simultaneo_Mx OR NOT #MEnt_DescargaAct),
                 PV := #V_CNTSeg_pHsMx,
                 BaseUnidades_ms := "CTE_BaseUnidades_1ms");
END_REGION

REGION Network 56: CONTADOR DE PRESENCIA - CNT_pHsMx
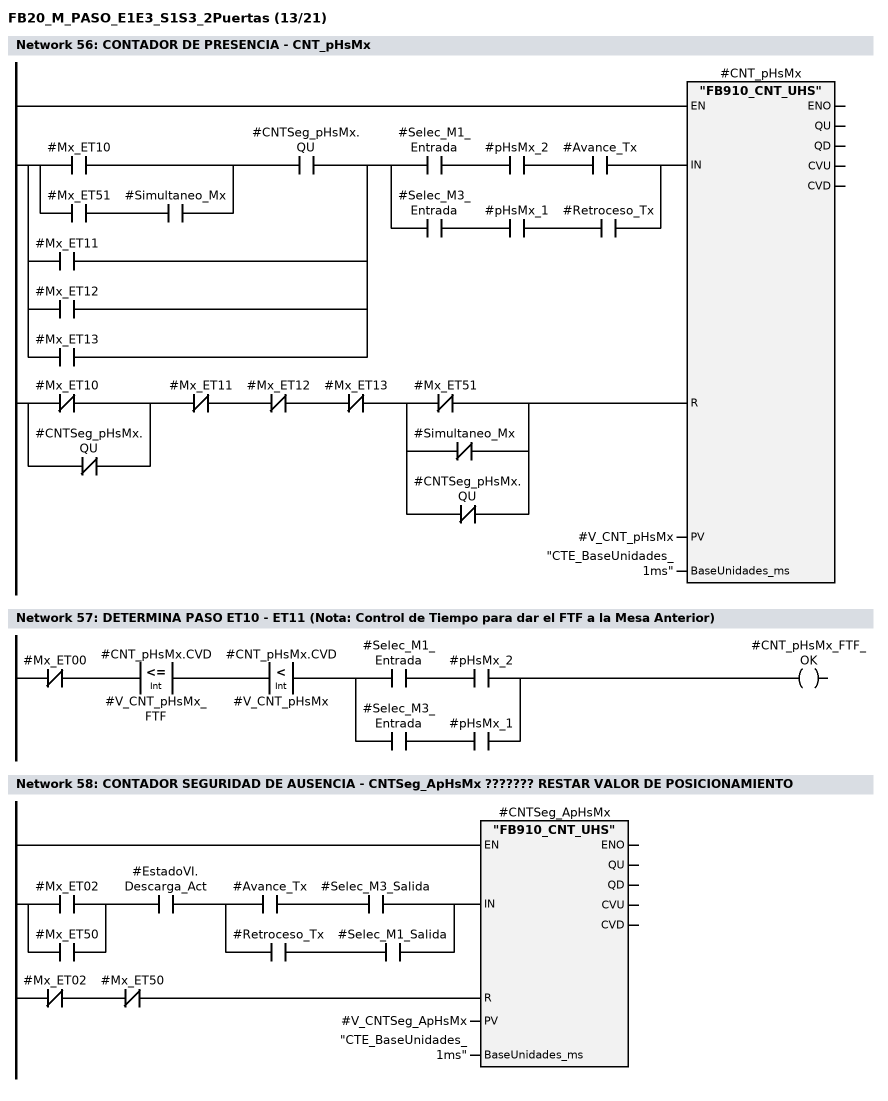
   RUNG wire#powerrail
      #CNT_pHsMx(IN := wire#w3, R := wire#w6, PV := #V_CNT_pHsMx, BaseUnidades_ms := "CTE_BaseUnidades_1ms", QU =>, QD =>, CVU =>, CVD =>)
   END_RUNG
   RUNG wire#powerrail
      Contact( #Mx_ET10 )
      wire#w1
      Contact( #CNTSeg_pHsMx.QU )
      wire#w2
      Contact( #Selec_M1_Entrada )
      Contact( #pHsMx_2 )
      Contact( #Avance_Tx )
   END_RUNG wire#w3
   RUNG wire#powerrail
      Contact( #Mx_ET51 )
      Contact( #Simultaneo_Mx )
   END_RUNG wire#w1
   RUNG wire#powerrail
      Contact( #Mx_ET11 )
   END_RUNG wire#w2
   RUNG wire#powerrail
      Contact( #Mx_ET12 )
   END_RUNG wire#w2
   RUNG wire#powerrail
      Contact( #Mx_ET13 )
   END_RUNG wire#w2
   RUNG wire#w2
      Contact( #Selec_M3_Entrada )
      Contact( #pHsMx_1 )
      Contact( #Retroceso_Tx )
   END_RUNG wire#w3
   RUNG wire#powerrail
      I_Contact( #Mx_ET10 )
      wire#w4
      I_Contact( #Mx_ET11 )
      I_Contact( #Mx_ET12 )
      I_Contact( #Mx_ET13 )
      wire#w5
      I_Contact( #Mx_ET51 )
   END_RUNG wire#w6
   RUNG wire#powerrail
      I_Contact( #CNTSeg_pHsMx.QU )
   END_RUNG wire#w4
   RUNG wire#w5
      I_Contact( #Simultaneo_Mx )
   END_RUNG wire#w6
   RUNG wire#w5
      I_Contact( #CNTSeg_pHsMx.QU )
   END_RUNG wire#w6
   // the same network as SCL:
   #CNT_pHsMx(IN := (((#Mx_ET10 OR (#Mx_ET51 AND #Simultaneo_Mx)) AND #CNTSeg_pHsMx.QU) OR #Mx_ET11 OR #Mx_ET12 OR #Mx_ET13) AND ((#Selec_M1_Entrada AND #pHsMx_2 AND #Avance_Tx) OR (#Selec_M3_Entrada AND #pHsMx_1 AND #Retroceso_Tx)),   // "FB910_CNT_UHS"
              R := (NOT #Mx_ET10 OR NOT #CNTSeg_pHsMx.QU) AND NOT #Mx_ET11 AND NOT #Mx_ET12 AND NOT #Mx_ET13 AND (NOT #Mx_ET51 OR NOT #Simultaneo_Mx OR NOT #CNTSeg_pHsMx.QU),
              PV := #V_CNT_pHsMx,
              BaseUnidades_ms := "CTE_BaseUnidades_1ms");
END_REGION

REGION Network 57: DETERMINA PASO ET10 - ET11 (Nota: Control de Tiempo para dar el FTF a la Mesa Anterior)
   RUNG wire#powerrail
      I_Contact( #Mx_ET00 )
      { S7_Templates := "SrcType := Int" } LE_Contact(in1 := #CNT_pHsMx.CVD, in2 := #V_CNT_pHsMx_FTF)
      { S7_Templates := "SrcType := Int" } LT_Contact(in1 := #CNT_pHsMx.CVD, in2 := #V_CNT_pHsMx)
      wire#w1
      Contact( #Selec_M1_Entrada )
      Contact( #pHsMx_2 )
      wire#w2
      Coil( #CNT_pHsMx_FTF_OK )
   END_RUNG
   RUNG wire#w1
      Contact( #Selec_M3_Entrada )
      Contact( #pHsMx_1 )
   END_RUNG wire#w2
   // the same network as SCL:
   #CNT_pHsMx_FTF_OK := NOT #Mx_ET00 AND (#CNT_pHsMx.CVD <= #V_CNT_pHsMx_FTF) AND (#CNT_pHsMx.CVD < #V_CNT_pHsMx) AND ((#Selec_M1_Entrada AND #pHsMx_2) OR (#Selec_M3_Entrada AND #pHsMx_1));
END_REGION

REGION Network 58: CONTADOR SEGURIDAD DE AUSENCIA - CNTSeg_ApHsMx ??????? RESTAR VALOR DE POSICIONAMIENTO
   RUNG wire#powerrail
      #CNTSeg_ApHsMx(IN := wire#w3, R := wire#w4, PV := #V_CNTSeg_ApHsMx, BaseUnidades_ms := "CTE_BaseUnidades_1ms", QU =>, QD =>, CVU =>, CVD =>)
   END_RUNG
   RUNG wire#powerrail
      Contact( #Mx_ET02 )
      wire#w1
      Contact( #EstadoVI.Descarga_Act )
      wire#w2
      Contact( #Avance_Tx )
      Contact( #Selec_M3_Salida )
   END_RUNG wire#w3
   RUNG wire#powerrail
      Contact( #Mx_ET50 )
   END_RUNG wire#w1
   RUNG wire#w2
      Contact( #Retroceso_Tx )
      Contact( #Selec_M1_Salida )
   END_RUNG wire#w3
   RUNG wire#powerrail
      I_Contact( #Mx_ET02 )
      I_Contact( #Mx_ET50 )
   END_RUNG wire#w4
   // the same network as SCL:
   #CNTSeg_ApHsMx(IN := (#Mx_ET02 OR #Mx_ET50) AND #EstadoVI.Descarga_Act AND ((#Avance_Tx AND #Selec_M3_Salida) OR (#Retroceso_Tx AND #Selec_M1_Salida)),   // "FB910_CNT_UHS"
                  R := NOT #Mx_ET02 AND NOT #Mx_ET50,
                  PV := #V_CNTSeg_ApHsMx,
                  BaseUnidades_ms := "CTE_BaseUnidades_1ms");
END_REGION

REGION Network 59: CONTADOR DE LA AUSENCIA - CNT_ApHsMX
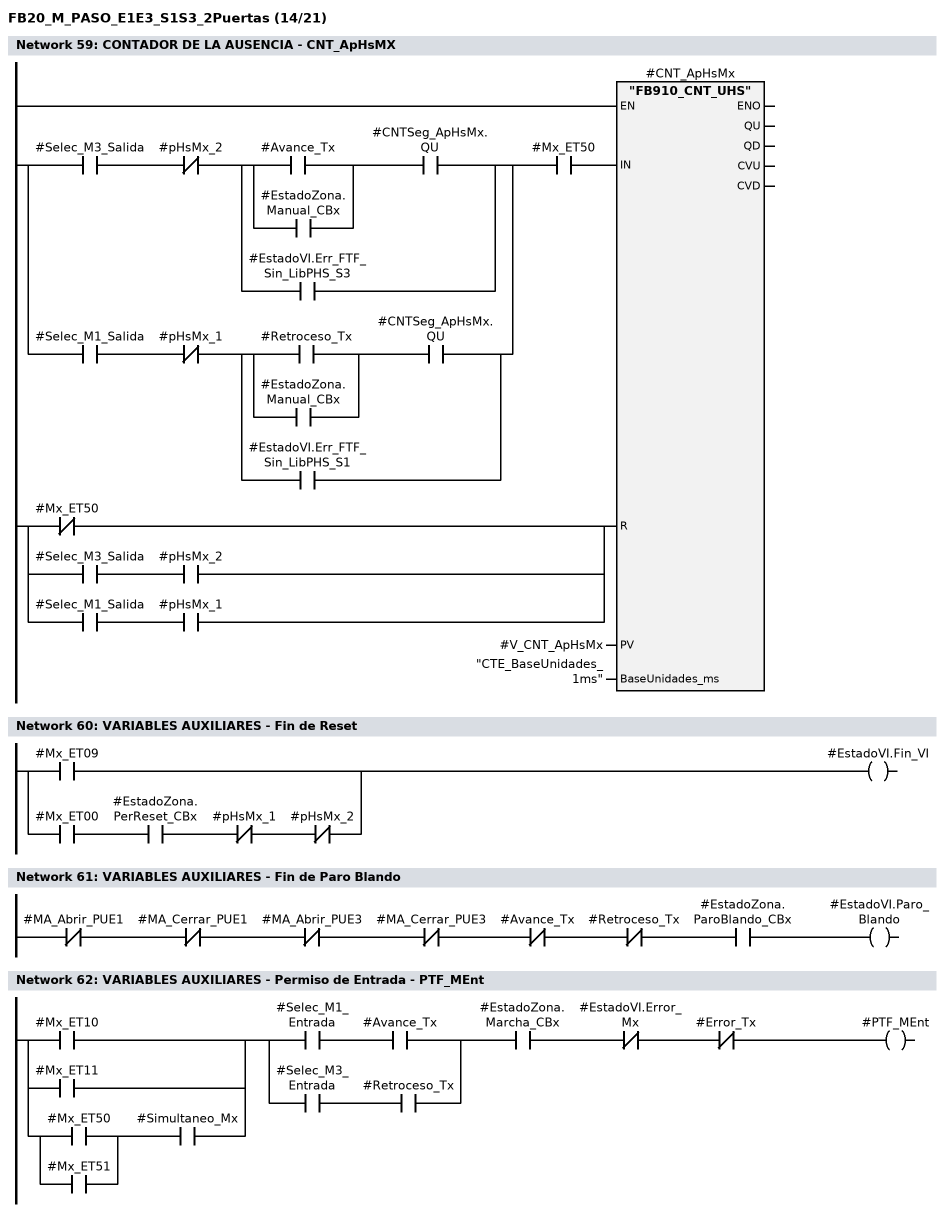
   RUNG wire#powerrail
      #CNT_ApHsMx(IN := wire#w6, R := wire#w7, PV := #V_CNT_ApHsMx, BaseUnidades_ms := "CTE_BaseUnidades_1ms", QU =>, QD =>, CVU =>, CVD =>)
   END_RUNG
   RUNG wire#powerrail
      Contact( #Selec_M3_Salida )
      I_Contact( #pHsMx_2 )
      wire#w1
      Contact( #Avance_Tx )
      wire#w2
      Contact( #CNTSeg_ApHsMx.QU )
      wire#w3
      Contact( #Mx_ET50 )
   END_RUNG wire#w6
   RUNG wire#w1
      Contact( #EstadoZona.Manual_CBx )
   END_RUNG wire#w2
   RUNG wire#w1
      Contact( #EstadoVI.Err_FTF_Sin_LibPHS_S3 )
   END_RUNG wire#w3
   RUNG wire#powerrail
      Contact( #Selec_M1_Salida )
      I_Contact( #pHsMx_1 )
      wire#w4
      Contact( #Retroceso_Tx )
      wire#w5
      Contact( #CNTSeg_ApHsMx.QU )
   END_RUNG wire#w3
   RUNG wire#w4
      Contact( #EstadoZona.Manual_CBx )
   END_RUNG wire#w5
   RUNG wire#w4
      Contact( #EstadoVI.Err_FTF_Sin_LibPHS_S1 )
   END_RUNG wire#w3
   RUNG wire#powerrail
      I_Contact( #Mx_ET50 )
   END_RUNG wire#w7
   RUNG wire#powerrail
      Contact( #Selec_M3_Salida )
      Contact( #pHsMx_2 )
   END_RUNG wire#w7
   RUNG wire#powerrail
      Contact( #Selec_M1_Salida )
      Contact( #pHsMx_1 )
   END_RUNG wire#w7
   // the same network as SCL:
   #CNT_ApHsMx(IN := ((#Selec_M3_Salida AND NOT #pHsMx_2 AND (((#Avance_Tx OR #EstadoZona.Manual_CBx) AND #CNTSeg_ApHsMx.QU) OR #EstadoVI.Err_FTF_Sin_LibPHS_S3)) OR (#Selec_M1_Salida AND NOT #pHsMx_1 AND (((#Retroceso_Tx OR #EstadoZona.Manual_CBx) AND #CNTSeg_ApHsMx.QU) OR #EstadoVI.Err_FTF_Sin_LibPHS_S1))) AND #Mx_ET50,   // "FB910_CNT_UHS"
               R := NOT #Mx_ET50 OR (#Selec_M3_Salida AND #pHsMx_2) OR (#Selec_M1_Salida AND #pHsMx_1),
               PV := #V_CNT_ApHsMx,
               BaseUnidades_ms := "CTE_BaseUnidades_1ms");
END_REGION

REGION Network 60: VARIABLES AUXILIARES - Fin de Reset
   RUNG wire#powerrail
      Contact( #Mx_ET09 )
      wire#w1
      Coil( #EstadoVI.Fin_VI )
   END_RUNG
   RUNG wire#powerrail
      Contact( #Mx_ET00 )
      Contact( #EstadoZona.PerReset_CBx )
      I_Contact( #pHsMx_1 )
      I_Contact( #pHsMx_2 )
   END_RUNG wire#w1
   // the same network as SCL:
   #EstadoVI.Fin_VI := #Mx_ET09 OR (#Mx_ET00 AND #EstadoZona.PerReset_CBx AND NOT #pHsMx_1 AND NOT #pHsMx_2);
END_REGION

REGION Network 61: VARIABLES AUXILIARES - Fin de Paro Blando
   RUNG wire#powerrail
      I_Contact( #MA_Abrir_PUE1 )
      I_Contact( #MA_Cerrar_PUE1 )
      I_Contact( #MA_Abrir_PUE3 )
      I_Contact( #MA_Cerrar_PUE3 )
      I_Contact( #Avance_Tx )
      I_Contact( #Retroceso_Tx )
      Contact( #EstadoZona.ParoBlando_CBx )
      Coil( #EstadoVI.Paro_Blando )
   END_RUNG
   // the same network as SCL:
   #EstadoVI.Paro_Blando := NOT #MA_Abrir_PUE1 AND NOT #MA_Cerrar_PUE1 AND NOT #MA_Abrir_PUE3 AND NOT #MA_Cerrar_PUE3 AND NOT #Avance_Tx AND NOT #Retroceso_Tx AND #EstadoZona.ParoBlando_CBx;
END_REGION

REGION Network 62: VARIABLES AUXILIARES - Permiso de Entrada - PTF_MEnt
   RUNG wire#powerrail
      Contact( #Mx_ET10 )
      wire#w1
      Contact( #Selec_M1_Entrada )
      Contact( #Avance_Tx )
      wire#w3
      Contact( #EstadoZona.Marcha_CBx )
      I_Contact( #EstadoVI.Error_Mx )
      I_Contact( #Error_Tx )
      Coil( #PTF_MEnt )
   END_RUNG
   RUNG wire#powerrail
      Contact( #Mx_ET11 )
   END_RUNG wire#w1
   RUNG wire#powerrail
      Contact( #Mx_ET50 )
      wire#w2
      Contact( #Simultaneo_Mx )
   END_RUNG wire#w1
   RUNG wire#powerrail
      Contact( #Mx_ET51 )
   END_RUNG wire#w2
   RUNG wire#w1
      Contact( #Selec_M3_Entrada )
      Contact( #Retroceso_Tx )
   END_RUNG wire#w3
   // the same network as SCL:
   #PTF_MEnt := (#Mx_ET10 OR #Mx_ET11 OR ((#Mx_ET50 OR #Mx_ET51) AND #Simultaneo_Mx)) AND ((#Selec_M1_Entrada AND #Avance_Tx) OR (#Selec_M3_Entrada AND #Retroceso_Tx)) AND #EstadoZona.Marcha_CBx AND NOT #EstadoVI.Error_Mx AND NOT #Error_Tx;
END_REGION

REGION Network 63: VARIABLES AUXILIARES - Aviso de Salida - AVTF_MSal
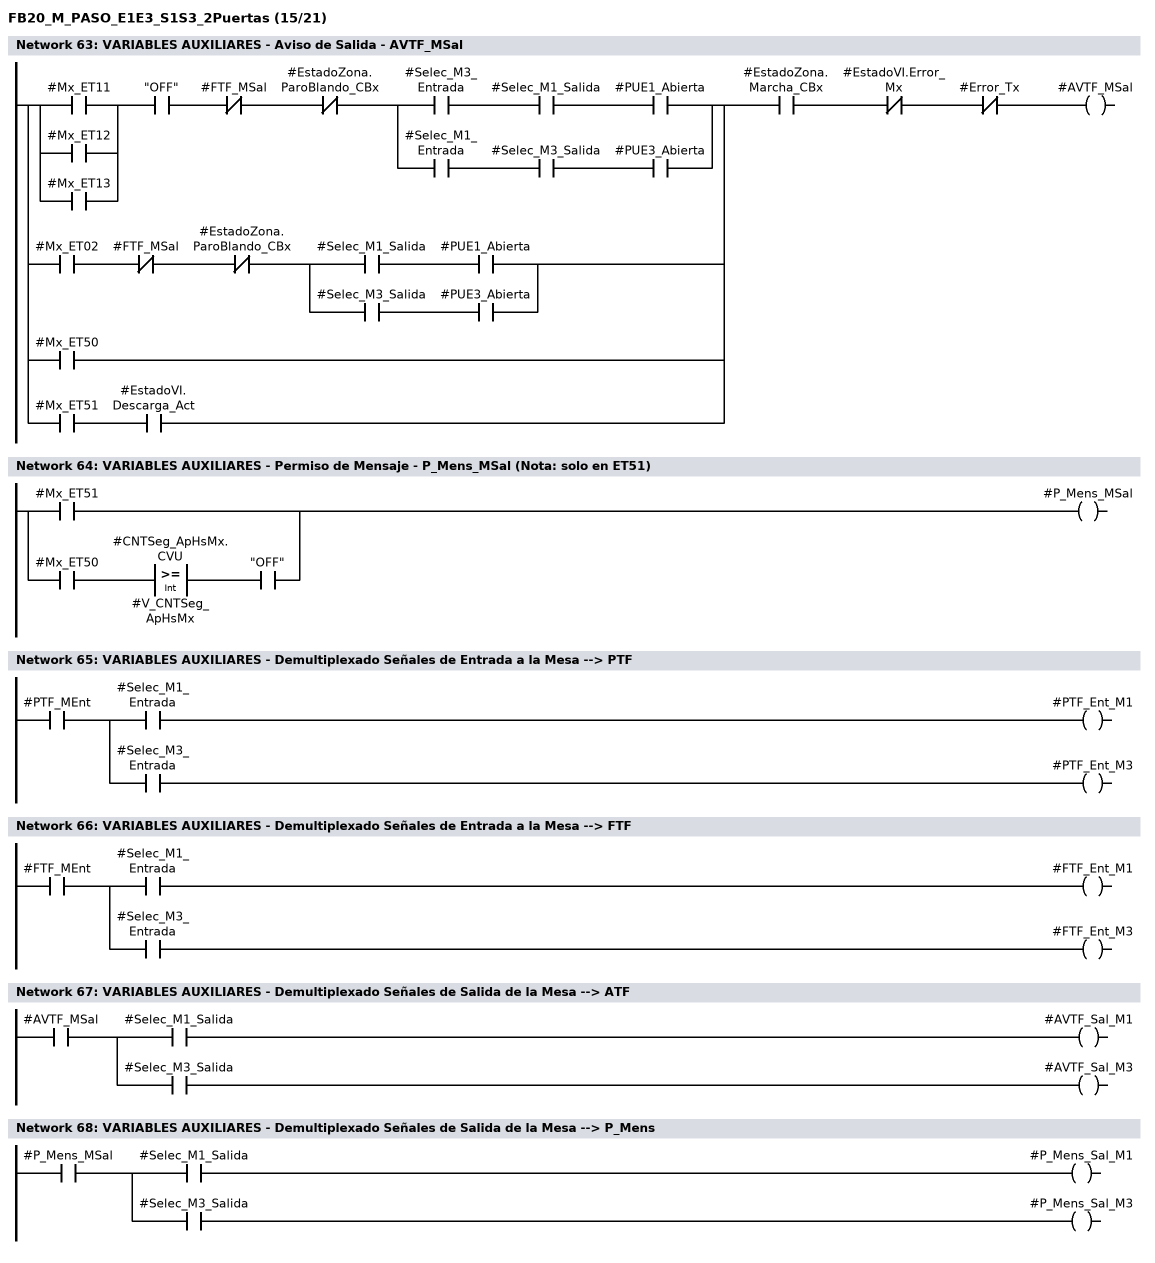
   RUNG wire#powerrail
      Contact( #Mx_ET11 )
      wire#w1
      Contact( "OFF" )
      I_Contact( #FTF_MSal )
      I_Contact( #EstadoZona.ParoBlando_CBx )
      wire#w2
      Contact( #Selec_M3_Entrada )
      Contact( #Selec_M1_Salida )
      Contact( #PUE1_Abierta )
      wire#w3
      Contact( #EstadoZona.Marcha_CBx )
      I_Contact( #EstadoVI.Error_Mx )
      I_Contact( #Error_Tx )
      Coil( #AVTF_MSal )
   END_RUNG
   RUNG wire#powerrail
      Contact( #Mx_ET12 )
   END_RUNG wire#w1
   RUNG wire#powerrail
      Contact( #Mx_ET13 )
   END_RUNG wire#w1
   RUNG wire#w2
      Contact( #Selec_M1_Entrada )
      Contact( #Selec_M3_Salida )
      Contact( #PUE3_Abierta )
   END_RUNG wire#w3
   RUNG wire#powerrail
      Contact( #Mx_ET02 )
      I_Contact( #FTF_MSal )
      I_Contact( #EstadoZona.ParoBlando_CBx )
      wire#w4
      Contact( #Selec_M1_Salida )
      Contact( #PUE1_Abierta )
   END_RUNG wire#w3
   RUNG wire#w4
      Contact( #Selec_M3_Salida )
      Contact( #PUE3_Abierta )
   END_RUNG wire#w3
   RUNG wire#powerrail
      Contact( #Mx_ET50 )
   END_RUNG wire#w3
   RUNG wire#powerrail
      Contact( #Mx_ET51 )
      Contact( #EstadoVI.Descarga_Act )
   END_RUNG wire#w3
   // the same network as SCL:
   #AVTF_MSal := (((#Mx_ET11 OR #Mx_ET12 OR #Mx_ET13) AND "OFF" AND NOT #FTF_MSal AND NOT #EstadoZona.ParoBlando_CBx AND ((#Selec_M3_Entrada AND #Selec_M1_Salida AND #PUE1_Abierta) OR (#Selec_M1_Entrada AND #Selec_M3_Salida AND #PUE3_Abierta))) OR (#Mx_ET02 AND NOT #FTF_MSal AND NOT #EstadoZona.ParoBlando_CBx AND ((#Selec_M1_Salida AND #PUE1_Abierta) OR (#Selec_M3_Salida AND #PUE3_Abierta))) OR #Mx_ET50 OR (#Mx_ET51 AND #EstadoVI.Descarga_Act)) AND #EstadoZona.Marcha_CBx AND NOT #EstadoVI.Error_Mx AND NOT #Error_Tx;
END_REGION

REGION Network 64: VARIABLES AUXILIARES - Permiso de Mensaje - P_Mens_MSal (Nota: solo en ET51)
   RUNG wire#powerrail
      Contact( #Mx_ET51 )
      wire#w1
      Coil( #P_Mens_MSal )
   END_RUNG
   RUNG wire#powerrail
      Contact( #Mx_ET50 )
      { S7_Templates := "SrcType := Int" } GE_Contact(in1 := #CNTSeg_ApHsMx.CVU, in2 := #V_CNTSeg_ApHsMx)
      Contact( "OFF" )
   END_RUNG wire#w1
   // the same network as SCL:
   #P_Mens_MSal := #Mx_ET51 OR (#Mx_ET50 AND (#CNTSeg_ApHsMx.CVU >= #V_CNTSeg_ApHsMx) AND "OFF");
END_REGION

REGION Network 65: VARIABLES AUXILIARES - Demultiplexado Señales de Entrada a la Mesa --> PTF
   RUNG wire#powerrail
      Contact( #PTF_MEnt )
      wire#w1
      Contact( #Selec_M1_Entrada )
      Coil( #PTF_Ent_M1 )
   END_RUNG
   RUNG wire#w1
      Contact( #Selec_M3_Entrada )
      Coil( #PTF_Ent_M3 )
   END_RUNG
   // the same network as SCL:
   #PTF_Ent_M1 := #PTF_MEnt AND #Selec_M1_Entrada;
   #PTF_Ent_M3 := #PTF_MEnt AND #Selec_M3_Entrada;
END_REGION

REGION Network 66: VARIABLES AUXILIARES - Demultiplexado Señales de Entrada a la Mesa --> FTF
   RUNG wire#powerrail
      Contact( #FTF_MEnt )
      wire#w1
      Contact( #Selec_M1_Entrada )
      Coil( #FTF_Ent_M1 )
   END_RUNG
   RUNG wire#w1
      Contact( #Selec_M3_Entrada )
      Coil( #FTF_Ent_M3 )
   END_RUNG
   // the same network as SCL:
   #FTF_Ent_M1 := #FTF_MEnt AND #Selec_M1_Entrada;
   #FTF_Ent_M3 := #FTF_MEnt AND #Selec_M3_Entrada;
END_REGION

REGION Network 67: VARIABLES AUXILIARES - Demultiplexado Señales de Salida de la Mesa --> ATF
   RUNG wire#powerrail
      Contact( #AVTF_MSal )
      wire#w1
      Contact( #Selec_M1_Salida )
      Coil( #AVTF_Sal_M1 )
   END_RUNG
   RUNG wire#w1
      Contact( #Selec_M3_Salida )
      Coil( #AVTF_Sal_M3 )
   END_RUNG
   // the same network as SCL:
   #AVTF_Sal_M1 := #AVTF_MSal AND #Selec_M1_Salida;
   #AVTF_Sal_M3 := #AVTF_MSal AND #Selec_M3_Salida;
END_REGION

REGION Network 68: VARIABLES AUXILIARES - Demultiplexado Señales de Salida de la Mesa --> P_Mens
   RUNG wire#powerrail
      Contact( #P_Mens_MSal )
      wire#w1
      Contact( #Selec_M1_Salida )
      Coil( #P_Mens_Sal_M1 )
   END_RUNG
   RUNG wire#w1
      Contact( #Selec_M3_Salida )
      Coil( #P_Mens_Sal_M3 )
   END_RUNG
   // the same network as SCL:
   #P_Mens_Sal_M1 := #P_Mens_MSal AND #Selec_M1_Salida;
   #P_Mens_Sal_M3 := #P_Mens_MSal AND #Selec_M3_Salida;
END_REGION

REGION Network 69: CONTADOR DE SIMULTANEO
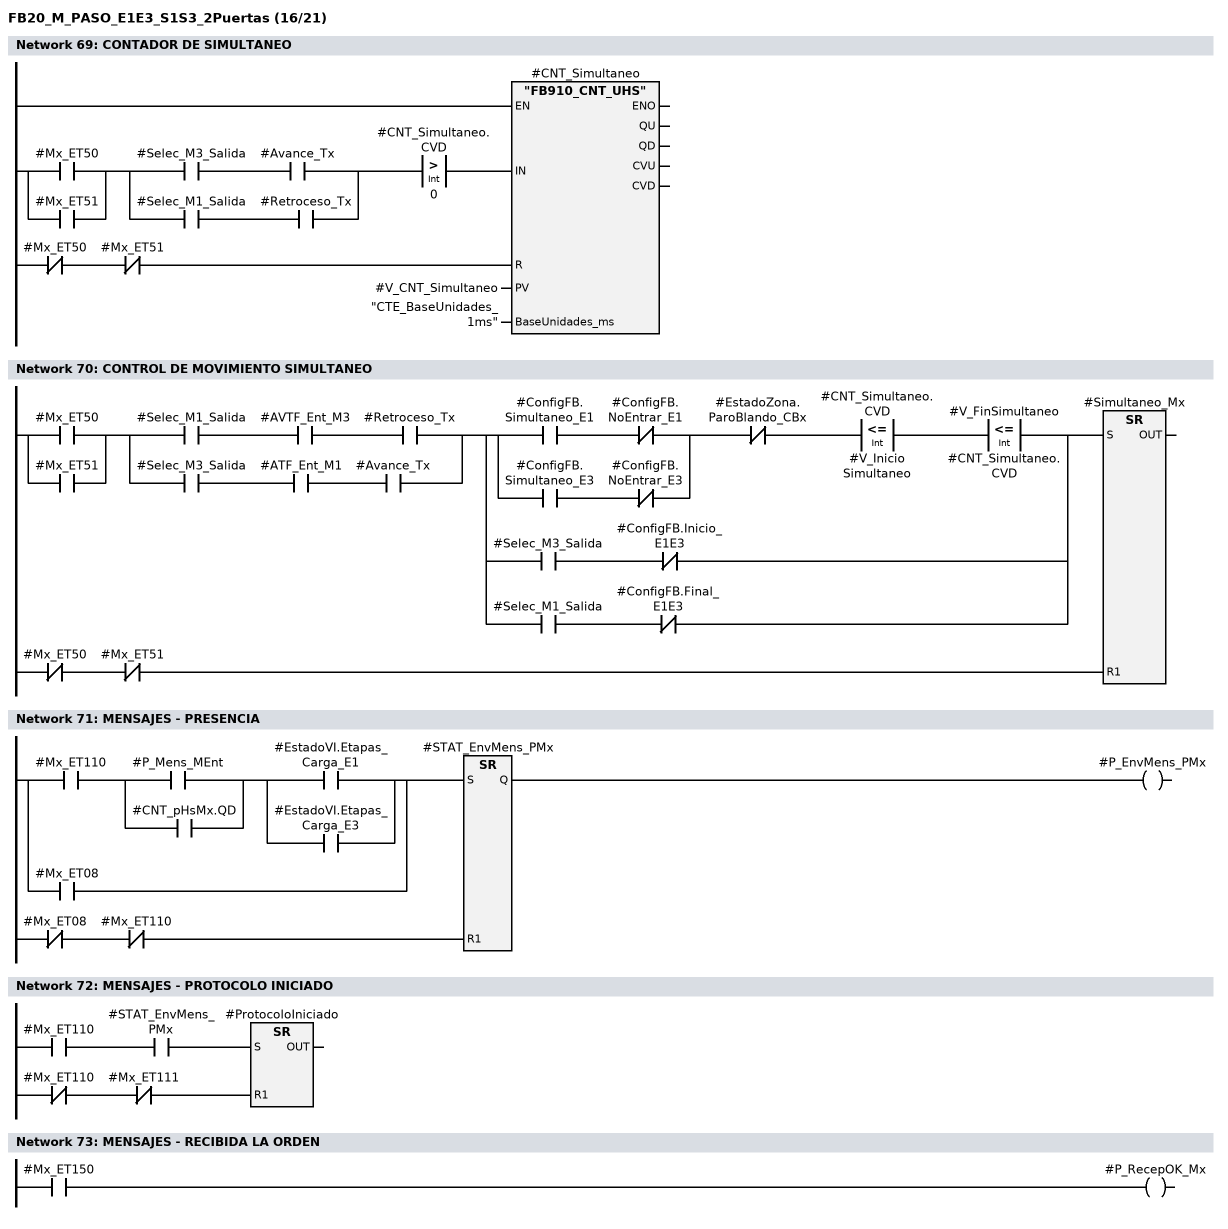
   RUNG wire#powerrail
      #CNT_Simultaneo(IN := wire#w3, R := wire#w4, PV := #V_CNT_Simultaneo, BaseUnidades_ms := "CTE_BaseUnidades_1ms", QU =>, QD =>, CVU =>, CVD =>)
   END_RUNG
   RUNG wire#powerrail
      Contact( #Mx_ET50 )
      wire#w1
      Contact( #Selec_M3_Salida )
      Contact( #Avance_Tx )
      wire#w2
      { S7_Templates := "SrcType := Int" } GT_Contact(in1 := #CNT_Simultaneo.CVD, in2 := 0)
   END_RUNG wire#w3
   RUNG wire#powerrail
      Contact( #Mx_ET51 )
   END_RUNG wire#w1
   RUNG wire#w1
      Contact( #Selec_M1_Salida )
      Contact( #Retroceso_Tx )
   END_RUNG wire#w2
   RUNG wire#powerrail
      I_Contact( #Mx_ET50 )
      I_Contact( #Mx_ET51 )
   END_RUNG wire#w4
   // the same network as SCL:
   #CNT_Simultaneo(IN := (#Mx_ET50 OR #Mx_ET51) AND ((#Selec_M3_Salida AND #Avance_Tx) OR (#Selec_M1_Salida AND #Retroceso_Tx)) AND (#CNT_Simultaneo.CVD > 0),   // "FB910_CNT_UHS"
                   R := NOT #Mx_ET50 AND NOT #Mx_ET51,
                   PV := #V_CNT_Simultaneo,
                   BaseUnidades_ms := "CTE_BaseUnidades_1ms");
END_REGION

REGION Network 70: CONTROL DE MOVIMIENTO SIMULTANEO
   RUNG wire#powerrail
      Contact( #Mx_ET50 )
      wire#w1
      Contact( #Selec_M1_Salida )
      Contact( #AVTF_Ent_M3 )
      Contact( #Retroceso_Tx )
      wire#w2
      Contact( #ConfigFB.Simultaneo_E1 )
      I_Contact( #ConfigFB.NoEntrar_E1 )
      wire#w3
      I_Contact( #EstadoZona.ParoBlando_CBx )
      { S7_Templates := "SrcType := Int" } LE_Contact(in1 := #CNT_Simultaneo.CVD, in2 := #V_InicioSimultaneo)
      { S7_Templates := "SrcType := Int" } LE_Contact(in1 := #V_FinSimultaneo, in2 := #CNT_Simultaneo.CVD)
      wire#w4
      S_SR(operand := #Simultaneo_Mx, r1 := wire#w5)
   END_RUNG
   RUNG wire#powerrail
      Contact( #Mx_ET51 )
   END_RUNG wire#w1
   RUNG wire#w1
      Contact( #Selec_M3_Salida )
      Contact( #ATF_Ent_M1 )
      Contact( #Avance_Tx )
   END_RUNG wire#w2
   RUNG wire#w2
      Contact( #ConfigFB.Simultaneo_E3 )
      I_Contact( #ConfigFB.NoEntrar_E3 )
   END_RUNG wire#w3
   RUNG wire#w2
      Contact( #Selec_M3_Salida )
      I_Contact( #ConfigFB.Inicio_E1E3 )
   END_RUNG wire#w4
   RUNG wire#w2
      Contact( #Selec_M1_Salida )
      I_Contact( #ConfigFB.Final_E1E3 )
   END_RUNG wire#w4
   RUNG wire#powerrail
      I_Contact( #Mx_ET50 )
      I_Contact( #Mx_ET51 )
   END_RUNG wire#w5
   // the same network as SCL:
   IF (#Mx_ET50 OR #Mx_ET51) AND ((#Selec_M1_Salida AND #AVTF_Ent_M3 AND #Retroceso_Tx) OR (#Selec_M3_Salida AND #ATF_Ent_M1 AND #Avance_Tx)) AND ((((#ConfigFB.Simultaneo_E1 AND NOT #ConfigFB.NoEntrar_E1) OR (#ConfigFB.Simultaneo_E3 AND NOT #ConfigFB.NoEntrar_E3)) AND NOT #EstadoZona.ParoBlando_CBx AND (#CNT_Simultaneo.CVD <= #V_InicioSimultaneo) AND (#V_FinSimultaneo <= #CNT_Simultaneo.CVD)) OR (#Selec_M3_Salida AND NOT #ConfigFB.Inicio_E1E3) OR (#Selec_M1_Salida AND NOT #ConfigFB.Final_E1E3)) THEN
       #Simultaneo_Mx := TRUE;   // SR flip-flop
   END_IF;
   IF NOT #Mx_ET50 AND NOT #Mx_ET51 THEN #Simultaneo_Mx := FALSE; END_IF;
END_REGION

REGION Network 71: MENSAJES - PRESENCIA
   RUNG wire#powerrail
      Contact( #Mx_ET110 )
      wire#w1
      Contact( #P_Mens_MEnt )
      wire#w2
      Contact( #EstadoVI.Etapas_Carga_E1 )
      wire#w3
      S_SR(operand := #STAT_EnvMens_PMx, r1 := wire#w4)
      Coil( #P_EnvMens_PMx )
   END_RUNG
   RUNG wire#w1
      Contact( #CNT_pHsMx.QD )
   END_RUNG wire#w2
   RUNG wire#w2
      Contact( #EstadoVI.Etapas_Carga_E3 )
   END_RUNG wire#w3
   RUNG wire#powerrail
      Contact( #Mx_ET08 )
   END_RUNG wire#w3
   RUNG wire#powerrail
      I_Contact( #Mx_ET08 )
      I_Contact( #Mx_ET110 )
   END_RUNG wire#w4
   // the same network as SCL:
   IF (#Mx_ET110 AND (#P_Mens_MEnt OR #CNT_pHsMx.QD) AND (#EstadoVI.Etapas_Carga_E1 OR #EstadoVI.Etapas_Carga_E3)) OR #Mx_ET08 THEN
       #STAT_EnvMens_PMx := TRUE;   // SR flip-flop
   END_IF;
   IF NOT #Mx_ET08 AND NOT #Mx_ET110 THEN #STAT_EnvMens_PMx := FALSE; END_IF;
   #P_EnvMens_PMx := #STAT_EnvMens_PMx;
END_REGION

REGION Network 72: MENSAJES - PROTOCOLO INICIADO
   RUNG wire#powerrail
      Contact( #Mx_ET110 )
      Contact( #STAT_EnvMens_PMx )
      S_SR(operand := #ProtocoloIniciado, r1 := wire#w1)
   END_RUNG
   RUNG wire#powerrail
      I_Contact( #Mx_ET110 )
      I_Contact( #Mx_ET111 )
   END_RUNG wire#w1
   // the same network as SCL:
   IF #Mx_ET110 AND #STAT_EnvMens_PMx THEN
       #ProtocoloIniciado := TRUE;   // SR flip-flop
   END_IF;
   IF NOT #Mx_ET110 AND NOT #Mx_ET111 THEN #ProtocoloIniciado := FALSE; END_IF;
END_REGION

REGION Network 73: MENSAJES - RECIBIDA LA ORDEN
   RUNG wire#powerrail
      Contact( #Mx_ET150 )
      Coil( #P_RecepOK_Mx )
   END_RUNG
   // the same network as SCL:
   #P_RecepOK_Mx := #Mx_ET150;
END_REGION

REGION Network 74: SALIDAS - Avance E1E3
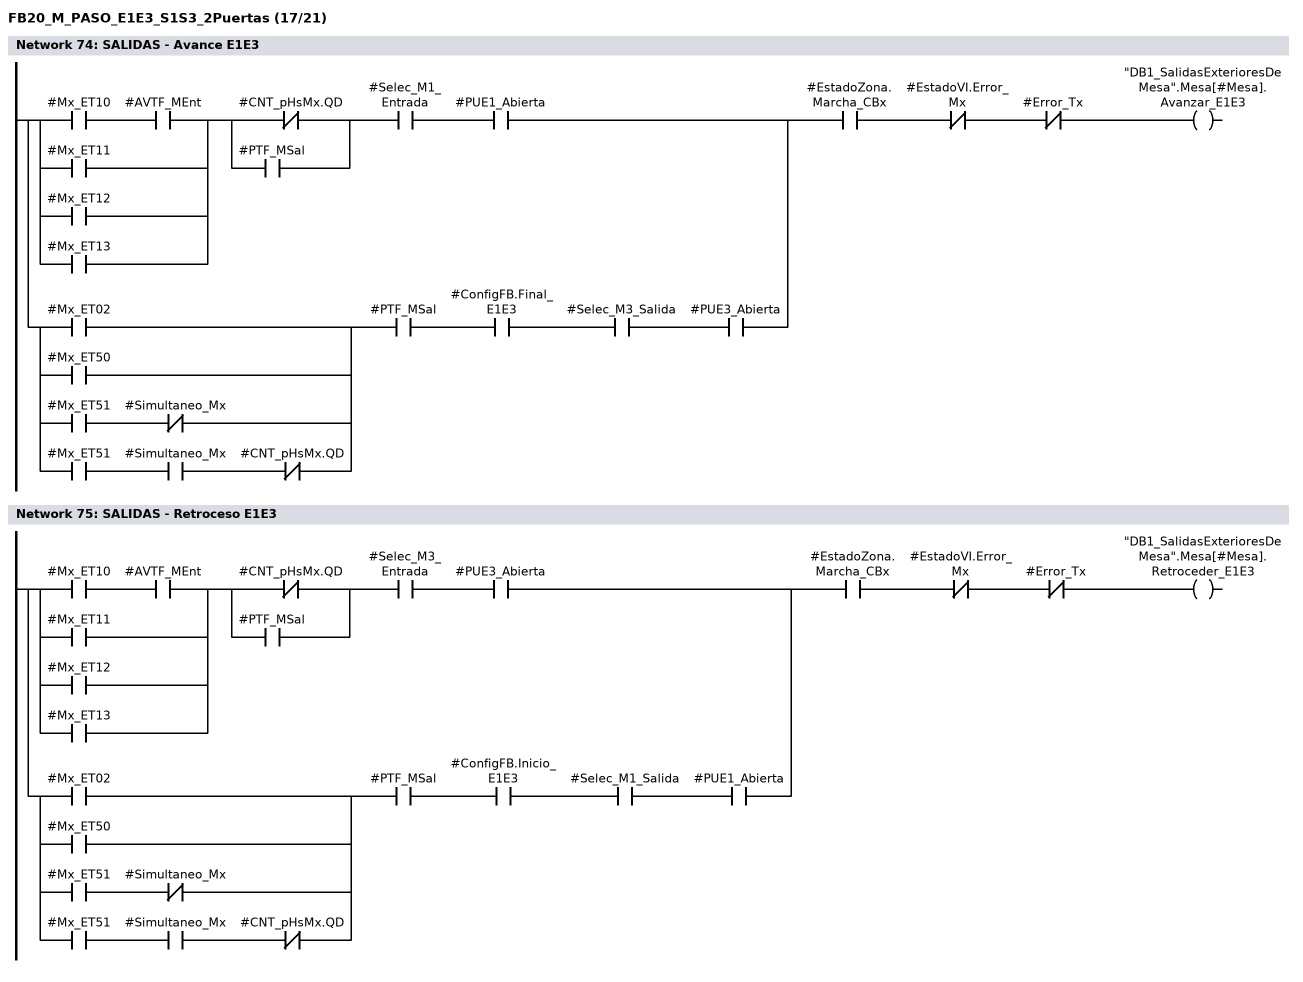
   RUNG wire#powerrail
      Contact( #Mx_ET10 )
      Contact( #AVTF_MEnt )
      wire#w1
      I_Contact( #CNT_pHsMx.QD )
      wire#w2
      Contact( #Selec_M1_Entrada )
      Contact( #PUE1_Abierta )
      wire#w3
      Contact( #EstadoZona.Marcha_CBx )
      I_Contact( #EstadoVI.Error_Mx )
      I_Contact( #Error_Tx )
      Coil( "DB1_SalidasExterioresDeMesa".Mesa[#Mesa].Avanzar_E1E3 )
   END_RUNG
   RUNG wire#powerrail
      Contact( #Mx_ET11 )
   END_RUNG wire#w1
   RUNG wire#powerrail
      Contact( #Mx_ET12 )
   END_RUNG wire#w1
   RUNG wire#powerrail
      Contact( #Mx_ET13 )
   END_RUNG wire#w1
   RUNG wire#w1
      Contact( #PTF_MSal )
   END_RUNG wire#w2
   RUNG wire#powerrail
      Contact( #Mx_ET02 )
      wire#w4
      Contact( #PTF_MSal )
      Contact( #ConfigFB.Final_E1E3 )
      Contact( #Selec_M3_Salida )
      Contact( #PUE3_Abierta )
   END_RUNG wire#w3
   RUNG wire#powerrail
      Contact( #Mx_ET50 )
   END_RUNG wire#w4
   RUNG wire#powerrail
      Contact( #Mx_ET51 )
      I_Contact( #Simultaneo_Mx )
   END_RUNG wire#w4
   RUNG wire#powerrail
      Contact( #Mx_ET51 )
      Contact( #Simultaneo_Mx )
      I_Contact( #CNT_pHsMx.QD )
   END_RUNG wire#w4
   // the same network as SCL:
   "DB1_SalidasExterioresDeMesa".Mesa[#Mesa].Avanzar_E1E3 := ((((#Mx_ET10 AND #AVTF_MEnt) OR #Mx_ET11 OR #Mx_ET12 OR #Mx_ET13) AND (NOT #CNT_pHsMx.QD OR #PTF_MSal) AND #Selec_M1_Entrada AND #PUE1_Abierta) OR ((#Mx_ET02 OR #Mx_ET50 OR (#Mx_ET51 AND NOT #Simultaneo_Mx) OR (#Mx_ET51 AND #Simultaneo_Mx AND NOT #CNT_pHsMx.QD)) AND #PTF_MSal AND #ConfigFB.Final_E1E3 AND #Selec_M3_Salida AND #PUE3_Abierta)) AND #EstadoZona.Marcha_CBx AND NOT #EstadoVI.Error_Mx AND NOT #Error_Tx;
END_REGION

REGION Network 75: SALIDAS - Retroceso E1E3
   RUNG wire#powerrail
      Contact( #Mx_ET10 )
      Contact( #AVTF_MEnt )
      wire#w1
      I_Contact( #CNT_pHsMx.QD )
      wire#w2
      Contact( #Selec_M3_Entrada )
      Contact( #PUE3_Abierta )
      wire#w3
      Contact( #EstadoZona.Marcha_CBx )
      I_Contact( #EstadoVI.Error_Mx )
      I_Contact( #Error_Tx )
      Coil( "DB1_SalidasExterioresDeMesa".Mesa[#Mesa].Retroceder_E1E3 )
   END_RUNG
   RUNG wire#powerrail
      Contact( #Mx_ET11 )
   END_RUNG wire#w1
   RUNG wire#powerrail
      Contact( #Mx_ET12 )
   END_RUNG wire#w1
   RUNG wire#powerrail
      Contact( #Mx_ET13 )
   END_RUNG wire#w1
   RUNG wire#w1
      Contact( #PTF_MSal )
   END_RUNG wire#w2
   RUNG wire#powerrail
      Contact( #Mx_ET02 )
      wire#w4
      Contact( #PTF_MSal )
      Contact( #ConfigFB.Inicio_E1E3 )
      Contact( #Selec_M1_Salida )
      Contact( #PUE1_Abierta )
   END_RUNG wire#w3
   RUNG wire#powerrail
      Contact( #Mx_ET50 )
   END_RUNG wire#w4
   RUNG wire#powerrail
      Contact( #Mx_ET51 )
      I_Contact( #Simultaneo_Mx )
   END_RUNG wire#w4
   RUNG wire#powerrail
      Contact( #Mx_ET51 )
      Contact( #Simultaneo_Mx )
      I_Contact( #CNT_pHsMx.QD )
   END_RUNG wire#w4
   // the same network as SCL:
   "DB1_SalidasExterioresDeMesa".Mesa[#Mesa].Retroceder_E1E3 := ((((#Mx_ET10 AND #AVTF_MEnt) OR #Mx_ET11 OR #Mx_ET12 OR #Mx_ET13) AND (NOT #CNT_pHsMx.QD OR #PTF_MSal) AND #Selec_M3_Entrada AND #PUE3_Abierta) OR ((#Mx_ET02 OR #Mx_ET50 OR (#Mx_ET51 AND NOT #Simultaneo_Mx) OR (#Mx_ET51 AND #Simultaneo_Mx AND NOT #CNT_pHsMx.QD)) AND #PTF_MSal AND #ConfigFB.Inicio_E1E3 AND #Selec_M1_Salida AND #PUE1_Abierta)) AND #EstadoZona.Marcha_CBx AND NOT #EstadoVI.Error_Mx AND NOT #Error_Tx;
END_REGION

REGION Network 76: SALIDAS - Parar E1E3
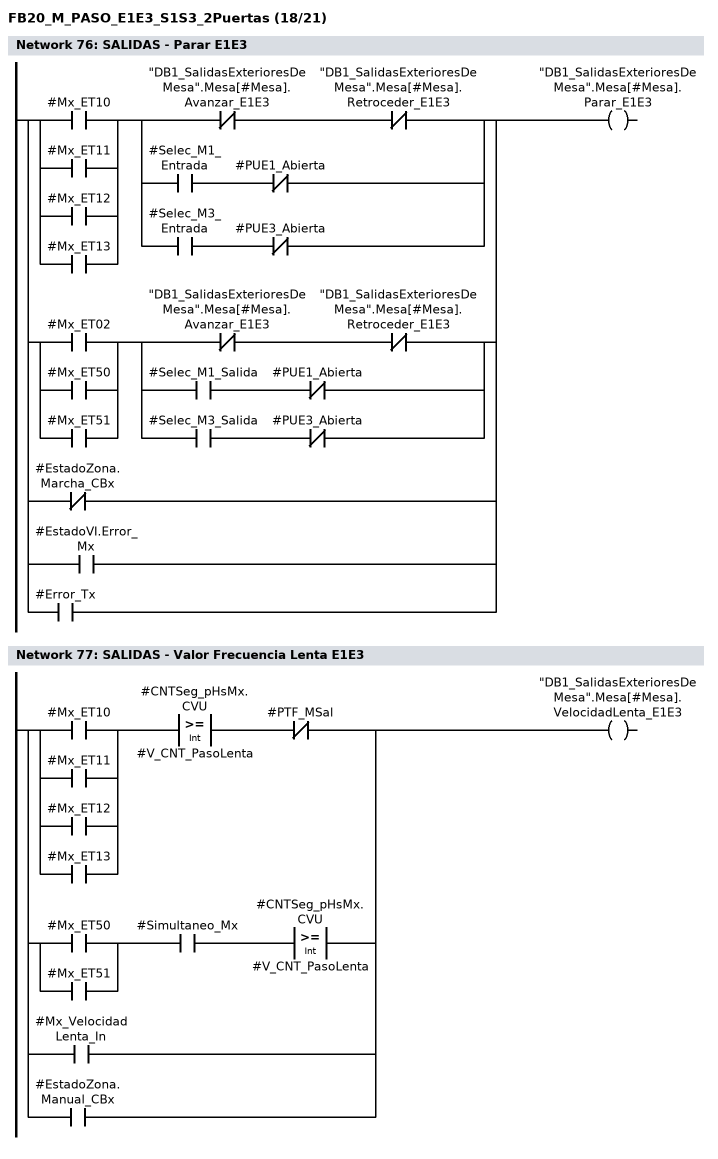
   RUNG wire#powerrail
      Contact( #Mx_ET10 )
      wire#w1
      I_Contact( "DB1_SalidasExterioresDeMesa".Mesa[#Mesa].Avanzar_E1E3 )
      I_Contact( "DB1_SalidasExterioresDeMesa".Mesa[#Mesa].Retroceder_E1E3 )
      wire#w2
      Coil( "DB1_SalidasExterioresDeMesa".Mesa[#Mesa].Parar_E1E3 )
   END_RUNG
   RUNG wire#powerrail
      Contact( #Mx_ET11 )
   END_RUNG wire#w1
   RUNG wire#powerrail
      Contact( #Mx_ET12 )
   END_RUNG wire#w1
   RUNG wire#powerrail
      Contact( #Mx_ET13 )
   END_RUNG wire#w1
   RUNG wire#w1
      Contact( #Selec_M1_Entrada )
      I_Contact( #PUE1_Abierta )
   END_RUNG wire#w2
   RUNG wire#w1
      Contact( #Selec_M3_Entrada )
      I_Contact( #PUE3_Abierta )
   END_RUNG wire#w2
   RUNG wire#powerrail
      Contact( #Mx_ET02 )
      wire#w3
      I_Contact( "DB1_SalidasExterioresDeMesa".Mesa[#Mesa].Avanzar_E1E3 )
      I_Contact( "DB1_SalidasExterioresDeMesa".Mesa[#Mesa].Retroceder_E1E3 )
   END_RUNG wire#w2
   RUNG wire#powerrail
      Contact( #Mx_ET50 )
   END_RUNG wire#w3
   RUNG wire#powerrail
      Contact( #Mx_ET51 )
   END_RUNG wire#w3
   RUNG wire#w3
      Contact( #Selec_M1_Salida )
      I_Contact( #PUE1_Abierta )
   END_RUNG wire#w2
   RUNG wire#w3
      Contact( #Selec_M3_Salida )
      I_Contact( #PUE3_Abierta )
   END_RUNG wire#w2
   RUNG wire#powerrail
      I_Contact( #EstadoZona.Marcha_CBx )
   END_RUNG wire#w2
   RUNG wire#powerrail
      Contact( #EstadoVI.Error_Mx )
   END_RUNG wire#w2
   RUNG wire#powerrail
      Contact( #Error_Tx )
   END_RUNG wire#w2
   // the same network as SCL:
   "DB1_SalidasExterioresDeMesa".Mesa[#Mesa].Parar_E1E3 := ((#Mx_ET10 OR #Mx_ET11 OR #Mx_ET12 OR #Mx_ET13) AND ((NOT "DB1_SalidasExterioresDeMesa".Mesa[#Mesa].Avanzar_E1E3 AND NOT "DB1_SalidasExterioresDeMesa".Mesa[#Mesa].Retroceder_E1E3) OR (#Selec_M1_Entrada AND NOT #PUE1_Abierta) OR (#Selec_M3_Entrada AND NOT #PUE3_Abierta))) OR ((#Mx_ET02 OR #Mx_ET50 OR #Mx_ET51) AND ((NOT "DB1_SalidasExterioresDeMesa".Mesa[#Mesa].Avanzar_E1E3 AND NOT "DB1_SalidasExterioresDeMesa".Mesa[#Mesa].Retroceder_E1E3) OR (#Selec_M1_Salida AND NOT #PUE1_Abierta) OR (#Selec_M3_Salida AND NOT #PUE3_Abierta))) OR NOT #EstadoZona.Marcha_CBx OR #EstadoVI.Error_Mx OR #Error_Tx;
END_REGION

REGION Network 77: SALIDAS - Valor Frecuencia Lenta E1E3
   RUNG wire#powerrail
      Contact( #Mx_ET10 )
      wire#w1
      { S7_Templates := "SrcType := Int" } GE_Contact(in1 := #CNTSeg_pHsMx.CVU, in2 := #V_CNT_PasoLenta)
      I_Contact( #PTF_MSal )
      wire#w2
      Coil( "DB1_SalidasExterioresDeMesa".Mesa[#Mesa].VelocidadLenta_E1E3 )
   END_RUNG
   RUNG wire#powerrail
      Contact( #Mx_ET11 )
   END_RUNG wire#w1
   RUNG wire#powerrail
      Contact( #Mx_ET12 )
   END_RUNG wire#w1
   RUNG wire#powerrail
      Contact( #Mx_ET13 )
   END_RUNG wire#w1
   RUNG wire#powerrail
      Contact( #Mx_ET50 )
      wire#w3
      Contact( #Simultaneo_Mx )
      { S7_Templates := "SrcType := Int" } GE_Contact(in1 := #CNTSeg_pHsMx.CVU, in2 := #V_CNT_PasoLenta)
   END_RUNG wire#w2
   RUNG wire#powerrail
      Contact( #Mx_ET51 )
   END_RUNG wire#w3
   RUNG wire#powerrail
      Contact( #Mx_VelocidadLenta_In )
   END_RUNG wire#w2
   RUNG wire#powerrail
      Contact( #EstadoZona.Manual_CBx )
   END_RUNG wire#w2
   // the same network as SCL:
   "DB1_SalidasExterioresDeMesa".Mesa[#Mesa].VelocidadLenta_E1E3 := ((#Mx_ET10 OR #Mx_ET11 OR #Mx_ET12 OR #Mx_ET13) AND (#CNTSeg_pHsMx.CVU >= #V_CNT_PasoLenta) AND NOT #PTF_MSal) OR ((#Mx_ET50 OR #Mx_ET51) AND #Simultaneo_Mx AND (#CNTSeg_pHsMx.CVU >= #V_CNT_PasoLenta)) OR #Mx_VelocidadLenta_In OR #EstadoZona.Manual_CBx;
END_REGION

REGION Network 78: SALIDAS - Abrir la PUERTA E1
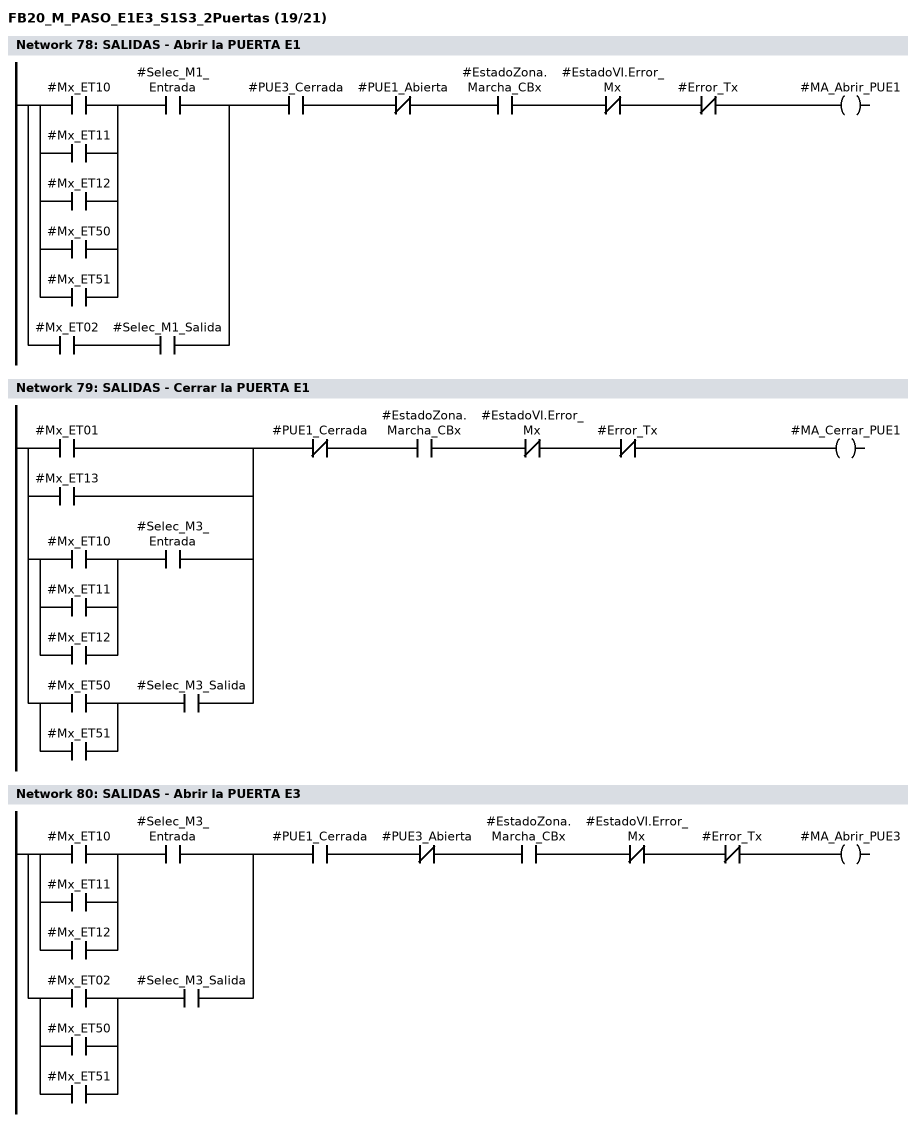
   RUNG wire#powerrail
      Contact( #Mx_ET10 )
      wire#w1
      Contact( #Selec_M1_Entrada )
      wire#w2
      Contact( #PUE3_Cerrada )
      I_Contact( #PUE1_Abierta )
      Contact( #EstadoZona.Marcha_CBx )
      I_Contact( #EstadoVI.Error_Mx )
      I_Contact( #Error_Tx )
      Coil( #MA_Abrir_PUE1 )
   END_RUNG
   RUNG wire#powerrail
      Contact( #Mx_ET11 )
   END_RUNG wire#w1
   RUNG wire#powerrail
      Contact( #Mx_ET12 )
   END_RUNG wire#w1
   RUNG wire#powerrail
      Contact( #Mx_ET50 )
   END_RUNG wire#w1
   RUNG wire#powerrail
      Contact( #Mx_ET51 )
   END_RUNG wire#w1
   RUNG wire#powerrail
      Contact( #Mx_ET02 )
      Contact( #Selec_M1_Salida )
   END_RUNG wire#w2
   // the same network as SCL:
   #MA_Abrir_PUE1 := (((#Mx_ET10 OR #Mx_ET11 OR #Mx_ET12 OR #Mx_ET50 OR #Mx_ET51) AND #Selec_M1_Entrada) OR (#Mx_ET02 AND #Selec_M1_Salida)) AND #PUE3_Cerrada AND NOT #PUE1_Abierta AND #EstadoZona.Marcha_CBx AND NOT #EstadoVI.Error_Mx AND NOT #Error_Tx;
END_REGION

REGION Network 79: SALIDAS - Cerrar la PUERTA E1
   RUNG wire#powerrail
      Contact( #Mx_ET01 )
      wire#w1
      I_Contact( #PUE1_Cerrada )
      Contact( #EstadoZona.Marcha_CBx )
      I_Contact( #EstadoVI.Error_Mx )
      I_Contact( #Error_Tx )
      Coil( #MA_Cerrar_PUE1 )
   END_RUNG
   RUNG wire#powerrail
      Contact( #Mx_ET13 )
   END_RUNG wire#w1
   RUNG wire#powerrail
      Contact( #Mx_ET10 )
      wire#w2
      Contact( #Selec_M3_Entrada )
   END_RUNG wire#w1
   RUNG wire#powerrail
      Contact( #Mx_ET11 )
   END_RUNG wire#w2
   RUNG wire#powerrail
      Contact( #Mx_ET12 )
   END_RUNG wire#w2
   RUNG wire#powerrail
      Contact( #Mx_ET50 )
      wire#w3
      Contact( #Selec_M3_Salida )
   END_RUNG wire#w1
   RUNG wire#powerrail
      Contact( #Mx_ET51 )
   END_RUNG wire#w3
   // the same network as SCL:
   #MA_Cerrar_PUE1 := (#Mx_ET01 OR #Mx_ET13 OR ((#Mx_ET10 OR #Mx_ET11 OR #Mx_ET12) AND #Selec_M3_Entrada) OR ((#Mx_ET50 OR #Mx_ET51) AND #Selec_M3_Salida)) AND NOT #PUE1_Cerrada AND #EstadoZona.Marcha_CBx AND NOT #EstadoVI.Error_Mx AND NOT #Error_Tx;
END_REGION

REGION Network 80: SALIDAS - Abrir la PUERTA E3
   RUNG wire#powerrail
      Contact( #Mx_ET10 )
      wire#w1
      Contact( #Selec_M3_Entrada )
      wire#w2
      Contact( #PUE1_Cerrada )
      I_Contact( #PUE3_Abierta )
      Contact( #EstadoZona.Marcha_CBx )
      I_Contact( #EstadoVI.Error_Mx )
      I_Contact( #Error_Tx )
      Coil( #MA_Abrir_PUE3 )
   END_RUNG
   RUNG wire#powerrail
      Contact( #Mx_ET11 )
   END_RUNG wire#w1
   RUNG wire#powerrail
      Contact( #Mx_ET12 )
   END_RUNG wire#w1
   RUNG wire#powerrail
      Contact( #Mx_ET02 )
      wire#w3
      Contact( #Selec_M3_Salida )
   END_RUNG wire#w2
   RUNG wire#powerrail
      Contact( #Mx_ET50 )
   END_RUNG wire#w3
   RUNG wire#powerrail
      Contact( #Mx_ET51 )
   END_RUNG wire#w3
   // the same network as SCL:
   #MA_Abrir_PUE3 := (((#Mx_ET10 OR #Mx_ET11 OR #Mx_ET12) AND #Selec_M3_Entrada) OR ((#Mx_ET02 OR #Mx_ET50 OR #Mx_ET51) AND #Selec_M3_Salida)) AND #PUE1_Cerrada AND NOT #PUE3_Abierta AND #EstadoZona.Marcha_CBx AND NOT #EstadoVI.Error_Mx AND NOT #Error_Tx;
END_REGION

REGION Network 81: SALIDAS - Cerrar la PUERTA E3
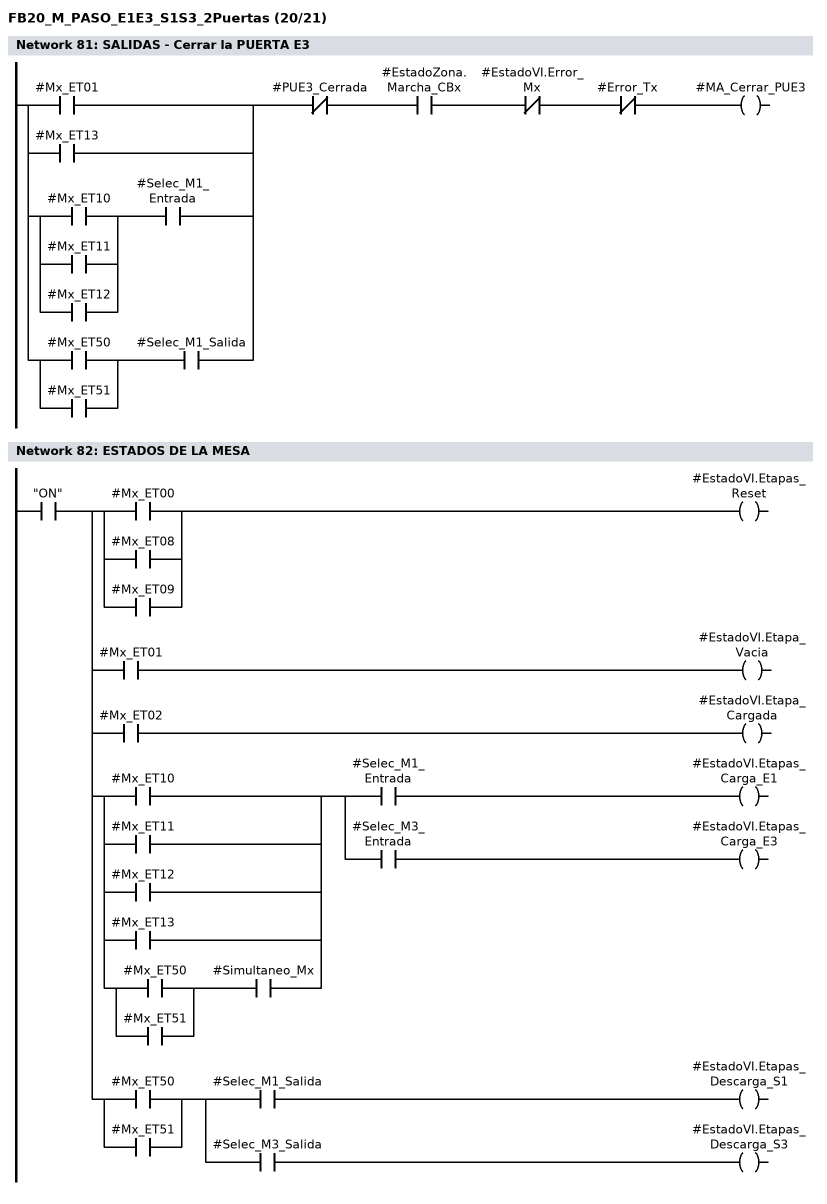
   RUNG wire#powerrail
      Contact( #Mx_ET01 )
      wire#w1
      I_Contact( #PUE3_Cerrada )
      Contact( #EstadoZona.Marcha_CBx )
      I_Contact( #EstadoVI.Error_Mx )
      I_Contact( #Error_Tx )
      Coil( #MA_Cerrar_PUE3 )
   END_RUNG
   RUNG wire#powerrail
      Contact( #Mx_ET13 )
   END_RUNG wire#w1
   RUNG wire#powerrail
      Contact( #Mx_ET10 )
      wire#w2
      Contact( #Selec_M1_Entrada )
   END_RUNG wire#w1
   RUNG wire#powerrail
      Contact( #Mx_ET11 )
   END_RUNG wire#w2
   RUNG wire#powerrail
      Contact( #Mx_ET12 )
   END_RUNG wire#w2
   RUNG wire#powerrail
      Contact( #Mx_ET50 )
      wire#w3
      Contact( #Selec_M1_Salida )
   END_RUNG wire#w1
   RUNG wire#powerrail
      Contact( #Mx_ET51 )
   END_RUNG wire#w3
   // the same network as SCL:
   #MA_Cerrar_PUE3 := (#Mx_ET01 OR #Mx_ET13 OR ((#Mx_ET10 OR #Mx_ET11 OR #Mx_ET12) AND #Selec_M1_Entrada) OR ((#Mx_ET50 OR #Mx_ET51) AND #Selec_M1_Salida)) AND NOT #PUE3_Cerrada AND #EstadoZona.Marcha_CBx AND NOT #EstadoVI.Error_Mx AND NOT #Error_Tx;
END_REGION

REGION Network 82: ESTADOS DE LA MESA
   RUNG wire#powerrail
      Contact( "ON" )
      wire#w1
      Contact( #Mx_ET00 )
      wire#w2
      Coil( #EstadoVI.Etapas_Reset )
   END_RUNG
   RUNG wire#w1
      Contact( #Mx_ET08 )
   END_RUNG wire#w2
   RUNG wire#w1
      Contact( #Mx_ET09 )
   END_RUNG wire#w2
   RUNG wire#w1
      Contact( #Mx_ET01 )
      Coil( #EstadoVI.Etapa_Vacia )
   END_RUNG
   RUNG wire#w1
      Contact( #Mx_ET02 )
      Coil( #EstadoVI.Etapa_Cargada )
   END_RUNG
   RUNG wire#w1
      Contact( #Mx_ET10 )
      wire#w3
      Contact( #Selec_M1_Entrada )
      Coil( #EstadoVI.Etapas_Carga_E1 )
   END_RUNG
   RUNG wire#w1
      Contact( #Mx_ET11 )
   END_RUNG wire#w3
   RUNG wire#w1
      Contact( #Mx_ET12 )
   END_RUNG wire#w3
   RUNG wire#w1
      Contact( #Mx_ET13 )
   END_RUNG wire#w3
   RUNG wire#w1
      Contact( #Mx_ET50 )
      wire#w4
      Contact( #Simultaneo_Mx )
   END_RUNG wire#w3
   RUNG wire#w1
      Contact( #Mx_ET51 )
   END_RUNG wire#w4
   RUNG wire#w3
      Contact( #Selec_M3_Entrada )
      Coil( #EstadoVI.Etapas_Carga_E3 )
   END_RUNG
   RUNG wire#w1
      Contact( #Mx_ET50 )
      wire#w5
      Contact( #Selec_M1_Salida )
      Coil( #EstadoVI.Etapas_Descarga_S1 )
   END_RUNG
   RUNG wire#w1
      Contact( #Mx_ET51 )
   END_RUNG wire#w5
   RUNG wire#w5
      Contact( #Selec_M3_Salida )
      Coil( #EstadoVI.Etapas_Descarga_S3 )
   END_RUNG
   // the same network as SCL:
   #EstadoVI.Etapas_Reset := "ON" AND (#Mx_ET00 OR #Mx_ET08 OR #Mx_ET09);
   #EstadoVI.Etapa_Vacia := "ON" AND #Mx_ET01;
   #EstadoVI.Etapa_Cargada := "ON" AND #Mx_ET02;
   #_w1 := "ON" AND (#Mx_ET10 OR #Mx_ET11 OR #Mx_ET12 OR #Mx_ET13 OR ((#Mx_ET50 OR #Mx_ET51) AND #Simultaneo_Mx));
   #EstadoVI.Etapas_Carga_E1 := #_w1 AND #Selec_M1_Entrada;
   #EstadoVI.Etapas_Carga_E3 := #_w1 AND #Selec_M3_Entrada;
   #_w2 := "ON" AND (#Mx_ET50 OR #Mx_ET51);
   #EstadoVI.Etapas_Descarga_S1 := #_w2 AND #Selec_M1_Salida;
   #EstadoVI.Etapas_Descarga_S3 := #_w2 AND #Selec_M3_Salida;
END_REGION

REGION Network 83: ENTRADAS DE LA MESA
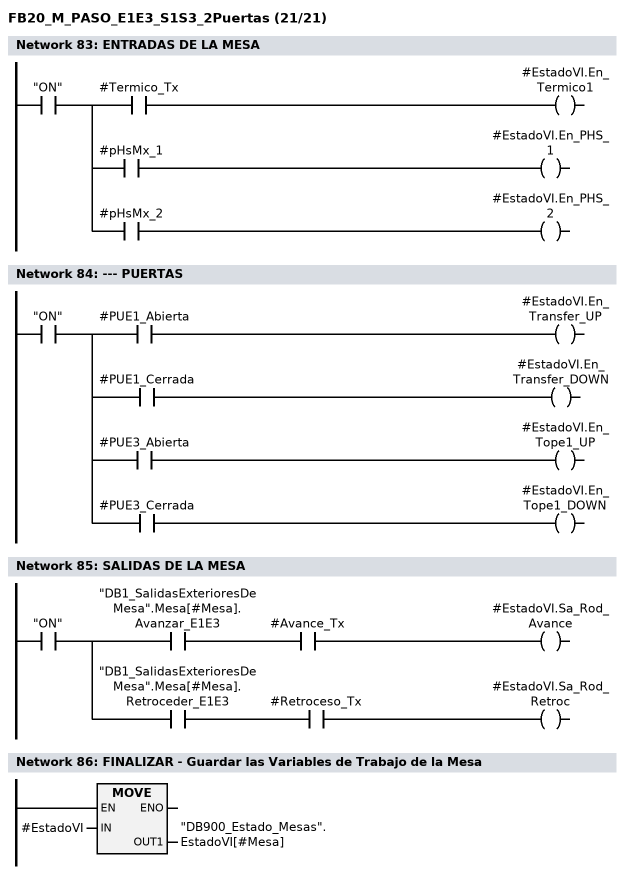
   RUNG wire#powerrail
      Contact( "ON" )
      wire#w1
      Contact( #Termico_Tx )
      Coil( #EstadoVI.En_Termico1 )
   END_RUNG
   RUNG wire#w1
      Contact( #pHsMx_1 )
      Coil( #EstadoVI.En_PHS_1 )
   END_RUNG
   RUNG wire#w1
      Contact( #pHsMx_2 )
      Coil( #EstadoVI.En_PHS_2 )
   END_RUNG
   // the same network as SCL:
   #EstadoVI.En_Termico1 := "ON" AND #Termico_Tx;
   #EstadoVI.En_PHS_1 := "ON" AND #pHsMx_1;
   #EstadoVI.En_PHS_2 := "ON" AND #pHsMx_2;
END_REGION

REGION Network 84: --- PUERTAS
   RUNG wire#powerrail
      Contact( "ON" )
      wire#w1
      Contact( #PUE1_Abierta )
      Coil( #EstadoVI.En_Transfer_UP )
   END_RUNG
   RUNG wire#w1
      Contact( #PUE1_Cerrada )
      Coil( #EstadoVI.En_Transfer_DOWN )
   END_RUNG
   RUNG wire#w1
      Contact( #PUE3_Abierta )
      Coil( #EstadoVI.En_Tope1_UP )
   END_RUNG
   RUNG wire#w1
      Contact( #PUE3_Cerrada )
      Coil( #EstadoVI.En_Tope1_DOWN )
   END_RUNG
   // the same network as SCL:
   #EstadoVI.En_Transfer_UP := "ON" AND #PUE1_Abierta;
   #EstadoVI.En_Transfer_DOWN := "ON" AND #PUE1_Cerrada;
   #EstadoVI.En_Tope1_UP := "ON" AND #PUE3_Abierta;
   #EstadoVI.En_Tope1_DOWN := "ON" AND #PUE3_Cerrada;
END_REGION

REGION Network 85: SALIDAS DE LA MESA
   RUNG wire#powerrail
      Contact( "ON" )
      wire#w1
      Contact( "DB1_SalidasExterioresDeMesa".Mesa[#Mesa].Avanzar_E1E3 )
      Contact( #Avance_Tx )
      Coil( #EstadoVI.Sa_Rod_Avance )
   END_RUNG
   RUNG wire#w1
      Contact( "DB1_SalidasExterioresDeMesa".Mesa[#Mesa].Retroceder_E1E3 )
      Contact( #Retroceso_Tx )
      Coil( #EstadoVI.Sa_Rod_Retroc )
   END_RUNG
   // the same network as SCL:
   #EstadoVI.Sa_Rod_Avance := "ON" AND "DB1_SalidasExterioresDeMesa".Mesa[#Mesa].Avanzar_E1E3 AND #Avance_Tx;
   #EstadoVI.Sa_Rod_Retroc := "ON" AND "DB1_SalidasExterioresDeMesa".Mesa[#Mesa].Retroceder_E1E3 AND #Retroceso_Tx;
END_REGION

REGION Network 86: FINALIZAR - Guardar las Variables de Trabajo de la Mesa
   RUNG wire#powerrail
      Move(in := #EstadoVI, out1 => "DB900_Estado_Mesas".EstadoVI[#Mesa])
   END_RUNG
   // the same network as SCL:
   "DB900_Estado_Mesas".EstadoVI[#Mesa] := #EstadoVI;
END_REGION
END_FUNCTION_BLOCK
